# B&R Automation Studio project BaseProject (part 3)

#### AdvIecChk.st - Implementation file
```iecst
(*****************************************************************************************************************************************
- This library is not officially supported by
- Just like IECCheck library, this library only works IF a programming error was caused in a
program written in IEC languages.
This library will NOT help TO troubleshoot pagefaults caused in C, C++ etc.
- Automation Runtime Simulation (ArSim) does NOT provide consistent backtrace with this
library.
- This library is capable OF catching many types OF IEC programming errors but NOT all.
[Example: IF a pointer is NOT a null pointer but it is just pointing TO an incorrect but
NOT invalid OR protected location in the memory. The memory copy operation using
such pointer might end up overwriting some part OF the memory.
When the processor tries TO ACCESS this corrupted memory location, it will cause a
pagefault. In such cases, the memory has already been corrupted, so there are no
ways TO tell what wrote into this memory.]
 *****************************************************************************************************************************************
 * Library: AdvIecCheck
 ****************************************************************************************************************************************
 ****************************************************************************************************************************************
 *																																		*
 * 							How	to	isolate	pagefaults	using	the	 AdvIecCheck	library?											*
 *							~~~~~~~~~~~~~~~~~~~~~~~~~~~~~~~~~~~~~~~~~~~~~~~~~~~~~~~~~~~~~~~~											*
 ****************************************************************************************************************************************
 ****************************************************************************************************************************************

			1 Overview

					1.1 What is a pagefault (Processor Exception Error)?
					 While a system is running, if the processor is commanded TO ACCESS an invalid OR protected
					memory location, it throws an exception TO the operating system. The B&R operating system logs
					these types OF serious memory violation errors as pagefaults.

					1.2 What can cause a pagefault?
					 Pagefaults can be caused BY programming errors AND sometimes it can be very difficult TO
					FIND the root cause OF it. The programming errors, such as incorrect reads OR writes can be caused BY
					following reasons:
					- Null OR incorrect pointer handle
					- Division BY zero
					- Invalid range OF enumeration
					- Invalid index ACCESS OF an array

					1.3 What is the difference between IECcheck & AdvIecCheck library?
					The IEC check library which is provided with Automation Studio checks division BY zero, null pointer,
					invalid array index, invalid enumeration range ACCESS AND invalid subrange.
					- IF IECcheck is NOT added TO a project, the checks FOR ‘null OR incorrect pointer handle, division
					BY zero, invalid range OF enumeration, and invalid index ACCESS OF an array’ are NOT
					performed, but when pagefault is encountered, you will get a backtrace.
					This backtrace may point you TO the line OF code that might have caused the pagefault.
					- IF IECcheck is added TO a project, the checks FOR ‘null OR incorrect pointer handle, division BY
					zero, invalid range OF enumeration, and invalid index ACCESS OF an array’ are performed.
					IF the processor finds any OF those checks TO be incorrect, a logbook error entry will inform
					you what type OF error were found AND which task class caused it, but you will get NOT get a
					backtrace.
					The Advance IEC Check library performs the same basic functions as IEC Check, but it also provides
					the following additional data about the location OF the pagefault.
					- Last executed task class cyclic
					- Last executed task’s name
					- Type OF programming error
					- Variable values from the last executed line OF code
					- Backtrace pointing TO the last executed line OF code

			2 Required Software
					- Automation Studio 4 (or higher)
					- Automation Runtime Embedded OR Automation Runtime Windows

			3 **************************************Warning****************************************************
			  **************************************Warning****************************************************
					- Just like IECCheck library, this library only works IF a programming error was caused in a
					program written in IEC languages.
					This library will NOT help TO troubleshoot pagefaults caused in C, C++ etc.
					- Automation Runtime Simulation (ArSim) does NOT provide consistent backtrace with this
					library.
					- This library is capable OF catching many types OF IEC programming errors but NOT all.
					[Example: IF a pointer is NOT a null pointer but it is just pointing TO an incorrect but
					NOT invalid OR protected location in the memory. The memory copy operation using
					such pointer might end up overwriting some part OF the memory.
					When the processor tries TO ACCESS this corrupted memory location, it will cause a
					pagefault. In such cases, the memory has already been corrupted, so there are no
					ways TO tell what wrote into this memory.]
			   **************************************Warning****************************************************
			   **************************************Warning****************************************************

			4 How TO use the AdvIecCheck Library?
			  How TO FIND the cause OF a pagefault?
					1. Unzip the attached AdvIecChk library.
					2. Add this library TO the Automation Studio project that is causing a pagefault.
					 Help on adding a user library can be found at:
					 Automation Studio Help > Programming > Libraries >
					 Example: Creating a user library> Exporting AND importing libraries
					3. Make sure the newly added AdvIecChk library is inside software configuration > library objects.
					4. Re-build the project AND transfer it TO the target OR create new compact flash card.
					5. Wait FOR the pagefaults.
					6. Try TO have multiple pagefaults & a repeatable way TO reproduce them before opening the logbook
					inside the project.
					7. Sort the logbook BY TIME.
					8. Warning entry will give you the following information about the pagefault trapped BY AdvIecChk.
					- Task class cyclic OF the task (E.g. task class 4)
					- Name OF the task (E.g. PageFault was the name OF my task)
					- Type OF programming error (E.g. Unsigned Subrange was outside valid range)
					- MAX, min valid value OF the variable that caused this fault
					(The valid range FOR that USINT was [3..20] AND the element the program was trying TO ACCESS
					was at location 0.)
					- Value OF the variable that ended up causing this fault
					9. Click on the Error entry AND go TO the backtrace, double click on the ‘FUNCTION start position’ OF the
					task name that you found inside the last warning message (It is ‘Pagefault’ in my example).
					Wherever the Automation Studio takes you, it is the line OF code where the pagefault was
					encountered.
					 10. After fixing the code, repeat the steps that you used TO cause the pagefault AND make sure the
					programing error is resolved.

			5 How TO disable IecCheck OR AdvIecCheck library in the project?
					IF the option -D _IGNORE_CHECKLIB is enabled in the additional build options, then the functions
					in this library are NOT used otherwise even IF you DELETE this library from software configuration,
					the compiler will use it.

			6 Best practices TO catch a pagefault
					Check FOR the following types OF operations:
					- Memory set, move, copy, and compare
					- String set, move, copy, and compare
					- Loop, enumeration AND array ranges
					- Use OF ADR(), ACCESS, and pointer handles TO FUNCTION blocks

			7 Additional note
					- You can customize AdvIecChk library TO get even more customized information out OF it
					- IF a non IEC language is causing pagefault, declare a remanent variable AND increase value OF
					that variable in your program. After a pagefault, you can connect TO the target AND read the
					value OF that remanent variable. Find out, at which point you set that value in your code.
					The programming error should be after that line OF code.

 ***************************************************************************************************************************************
 ******************************************************Release Notes********************************************************************
Revision 1.00.0    - Matt Buck & Matt Adams
- Started distributing from 2013
- Better logger entries
 ******************************************************************************************************************************************
Revision 2.00.0    - Varad Darji
- Started distributing from Automation Conf. 2015
- Improvement for logger entries
- Provides backtrace
- gIecChkSec entries does NOT need TO be part OF this code there anymore because we are getting an actual backtrace now.
  They are there for legacy reasons.
- Created new documentation & added it to the library as well.
 ******************************************************************************************************************************************
 ******************************************************************************************************************************************)

(* Check divisor for DINT and UDINT division *)
FUNCTION CheckDivDWord
	IF divisor=0 THEN
		CheckDivDWord:=1;
		MakeEntry(55555,divisor,'Divide by Zero - Double Word');

		//Note: DarjiV, creating a pagefault on purpose to get the backtrace data
		//				This function does not provide consistant back
		memcpy(1,1,1);

	ELSE
		CheckDivDWord:=divisor;
	END_IF
END_FUNCTION

(* Check divisor for INT and UINT division *)
FUNCTION CheckDivWord
	IF divisor=0 THEN
		CheckDivWord:=1;
		MakeEntry(55555,divisor,'Divide by Zero - Word');

		//creating a pagefault on purpose to get the backtrace data
		memcpy(1,1,1);
	ELSE
		CheckDivWord:=divisor;
	END_IF
END_FUNCTION

(* Check divisor for SINT and USINT division *)
FUNCTION CheckDivByte
	IF divisor=0 THEN
		CheckDivByte:=1;
		MakeEntry(55555,divisor,'Divide by Zero - Byte');

		//creating a pagefault on purpose to get the backtrace data
		memcpy(1,1,1);
	ELSE
		CheckDivByte:=divisor;
	END_IF
END_FUNCTION

(* Check divisor for REAL division *)
FUNCTION CheckDivReal
	IF divisor=0 THEN
		CheckDivReal:=1;
		MakeEntry(55555,0,'Divide by Zero - Real');

		//creating a pagefault on purpose to get the backtrace data
		memcpy(1,1,1);
	ELSE
		CheckDivReal:=divisor;
	END_IF
END_FUNCTION

(* Check divisor for LREAL division *)
FUNCTION CheckDivLReal
	IF divisor=0 THEN
		CheckDivLReal:=1;
		MakeEntry(55555,0,'Divide by Zero - Long Real');

		//creating a pagefault on purpose to get the backtrace data
		memcpy(1,1,1);
	ELSE
		CheckDivLReal:=divisor;
	END_IF
END_FUNCTION

(* Check range for enumeration *)
FUNCTION CheckRange
	IF value < lower THEN
		CheckRange := lower;

		itoa(lower, ADR(LowString));
		itoa(upper, ADR(UpString));
		itoa(value, ADR(IndexString));
		strcpy(ADR(text),ADR('ENUM-Check Low. Value '));
		strcat(ADR(text),ADR(IndexString));
		strcat(ADR(text),ADR(' is outside ['));
		strcat(ADR(text),ADR(LowString));
		strcat(ADR(text),ADR('..'));
		strcat(ADR(text),ADR(UpString));
		strcat(ADR(text),ADR(']'));
		MakeEntry(55555,value,text);
		//creating a pagefault on purpose to get the backtrace data
		memcpy(1,1,1);

	ELSIF value > upper THEN
		CheckRange := upper;

		itoa(lower, ADR(LowString));
		itoa(upper, ADR(UpString));
		itoa(value, ADR(IndexString));
		strcpy(ADR(text),ADR('ENUM-Check High. Value '));
		strcat(ADR(text),ADR(IndexString));
		strcat(ADR(text),ADR(' is outside ['));
		strcat(ADR(text),ADR(LowString));
		strcat(ADR(text),ADR('..'));
		strcat(ADR(text),ADR(UpString));
		strcat(ADR(text),ADR(']'));
		MakeEntry(55555,value,text);
		//creating a pagefault on purpose to get the backtrace data
		memcpy(1,1,1);
	ELSE
		CheckRange := value;
	END_IF
END_FUNCTION

(* Check range for subrange of signed data types *)
FUNCTION CheckSignedSubrange
	IF value < lower THEN
		CheckSignedSubrange := lower;

		itoa(lower, ADR(LowString));
		itoa(upper, ADR(UpString));
		itoa(value, ADR(IndexString));
		strcpy(ADR(text),ADR('Signed Subrange Index '));
		strcat(ADR(text),ADR(IndexString));
		strcat(ADR(text),ADR(' is outside ['));
		strcat(ADR(text),ADR(LowString));
		strcat(ADR(text),ADR('..'));
		strcat(ADR(text),ADR(UpString));
		strcat(ADR(text),ADR(']'));
		MakeEntry(55555,value,text);
		//creating a pagefault on purpose to get the backtrace data
		memcpy(1,1,1);

	ELSIF value > upper THEN
		CheckSignedSubrange := upper;

		itoa(lower, ADR(LowString));
		itoa(upper, ADR(UpString));
		itoa(value, ADR(IndexString));
		strcpy(ADR(text),ADR('Signed Subrange Index '));
		strcat(ADR(text),ADR(IndexString));
		strcat(ADR(text),ADR(' is outside ['));
		strcat(ADR(text),ADR(LowString));
		strcat(ADR(text),ADR('..'));
		strcat(ADR(text),ADR(UpString));
		strcat(ADR(text),ADR(']'));
		MakeEntry(55555,value,text);
		//creating a pagefault on purpose to get the backtrace data
		memcpy(1,1,1);
	ELSE
		CheckSignedSubrange := value;
	END_IF
END_FUNCTION

(* Check range for subrange of unsigned data types *)
FUNCTION CheckUnsignedSubrange
	IF value < lower THEN
		CheckUnsignedSubrange := lower;

		itoa(lower, ADR(LowString));
		itoa(upper, ADR(UpString));
		itoa(value, ADR(IndexString));
		strcpy(ADR(text),ADR('Unsigned Subrange Index '));
		strcat(ADR(text),ADR(IndexString));
		strcat(ADR(text),ADR(' is outside ['));
		strcat(ADR(text),ADR(LowString));
		strcat(ADR(text),ADR('..'));
		strcat(ADR(text),ADR(UpString));
		strcat(ADR(text),ADR(']'));
		MakeEntry(55555,value,text);
		//creating a pagefault on purpose to get the backtrace data
		memcpy(1,1,1);

	ELSIF value > upper THEN
		CheckUnsignedSubrange := upper;

		itoa(lower, ADR(LowString));
		itoa(upper, ADR(UpString));
		itoa(value, ADR(IndexString));
		strcpy(ADR(text),ADR('Unsigned Subrange Index '));
		strcat(ADR(text),ADR(IndexString));
		strcat(ADR(text),ADR(' is outside ['));
		strcat(ADR(text),ADR(LowString));
		strcat(ADR(text),ADR('..'));
		strcat(ADR(text),ADR(UpString));
		strcat(ADR(text),ADR(']'));
		MakeEntry(55555,value,text);
		//creating a pagefault on purpose to get the backtrace data
		memcpy(1,1,1);
	ELSE
		CheckUnsignedSubrange := value;
	END_IF
END_FUNCTION

(* Check address when reading dynamic variables *)
FUNCTION CheckReadAccess
	IF address=0 THEN
		(* TODO: Insert an appropriate code, see AutomationStudio help for further information *)
		MakeEntry(55555,address,'Attempt to read from address of zero / NULL');
		//creating a pagefault on purpose to get the backtrace data
		memcpy(1,1,1);

	END_IF

	CheckReadAccess:=0;
END_FUNCTION

(* Check address when writing dynamic variables *)
FUNCTION CheckWriteAccess
	IF address=0 THEN
		(* TODO: Insert an appropriate code, see AutomationStudio help for further information *)
		MakeEntry(55555,address,'Attempt to write to address of zero / NULL');
		//creating a pagefault on purpose to get the backtrace data
		memcpy(1,1,1);
	END_IF

	CheckWriteAccess:=0;
END_FUNCTION

FUNCTION CheckBounds (* Check range for array access *)
	IF index < lower OR index > upper THEN
		itoa(lower, ADR(LowString));
		itoa(upper, ADR(UpString));
		itoa(index, ADR(IndexString));
		CheckBounds := upper;
		strcpy(ADR(text),ADR('Array Index '));
		strcat(ADR(text),ADR(IndexString));
		strcat(ADR(text),ADR(' is outside ['));
		strcat(ADR(text),ADR(LowString));
		strcat(ADR(text),ADR('..'));
		strcat(ADR(text),ADR(UpString));
		strcat(ADR(text),ADR(']'));
		MakeEntry(55555,index,text);
		//creating a pagefault on purpose to get the backtrace data
		memcpy(1,1,1);
	ELSE
		CheckBounds := index;
	END_IF
END_FUNCTION

FUNCTION MakeEntry (* Makes a log book entry. Note that gIecChkSec must be a global DINT! *)
	status_name := ST_name(0,ADR(taskname),ADR(group));
	PV_xgetadr(ADR('gIecChkSec'), ADR(pv_adr), ADR(data_len));
	IF pv_adr > 0 AND data_len > 0 THEN
		memcpy(ADR(SectionData),pv_adr,data_len);
		itoa(SectionData,ADR(SectionString));
	END_IF

	strcpy(ADR(out_text),ADR(text));
	strcat(ADR(out_text),ADR(' in task "'));
	strcat(ADR(out_text),ADR(taskname));
	strcat(ADR(out_text),ADR('" Section:'));
	strcat(ADR(out_text),ADR(SectionString));
	MakeEntry := ADR(out_text);

	// Making Logger entry & restarting
	ERRxwarning(number,index,ADR(out_text));
	// Change Note DarjiV: Change ERRxfatel_FB to ERRxwarning_FB because to get additional data.
	// 						Because I want TO finish this function and go back TO whichever function started this function and cause a pagefault there to get backtrace to the CODE.
	//						Now the AdvanceIEC Check library will give a pagefault location in CODE & the values of those variable when the pagefault happened.

END_FUNCTION
```

### Program Logical/Source/GlobalSetup (IEC)

#### Main.st
```iecst
PROGRAM _INIT
	(* Call global variables until they are use somewhere else *)
	gSampleTrak;
	gSampleTrak_SectorTrakA;
	gSampleTrak_SectorTrakB;
	gSampleTrak_SectorTrakAll;
	gSampleTrakMon;

	#ifdef ASSEMBLY_STANDARD
	(*All segment references must be included in the following segment array*)
	gTrakData.Seg.SegList[0].Name  := 'gSeg_A_1'; 		gTrakData.Seg.SegList[0].McType := gSeg_A_1 ;
	gTrakData.Seg.SegList[1].Name  := 'gSeg_A_2';		gTrakData.Seg.SegList[1].McType := gSeg_A_2 ;
	gTrakData.Seg.SegList[2].Name  := 'gSeg_A_3'; 		gTrakData.Seg.SegList[2].McType := gSeg_A_3 ;
	gTrakData.Seg.SegList[3].Name  := 'gSeg_A_4';		gTrakData.Seg.SegList[3].McType := gSeg_A_4 ;
	gTrakData.Seg.SegList[4].Name  := 'gSeg_A_5';		gTrakData.Seg.SegList[4].McType := gSeg_A_5 ;
	gTrakData.Seg.SegList[5].Name  := 'gSeg_A_6';		gTrakData.Seg.SegList[5].McType := gSeg_A_6 ;
	gTrakData.Seg.SegList[6].Name  := 'gSeg_A_7';		gTrakData.Seg.SegList[6].McType := gSeg_A_7 ;
	gTrakData.Seg.SegList[7].Name  := 'gSeg_A_8';		gTrakData.Seg.SegList[7].McType := gSeg_A_8 ;
	gTrakData.Seg.SegList[8].Name  := 'gSeg_A_9';		gTrakData.Seg.SegList[8].McType := gSeg_A_9 ;
	gTrakData.Seg.SegList[9].Name  := 'gSeg_A_10';		gTrakData.Seg.SegList[9].McType := gSeg_A_10;
	gTrakData.Seg.SegList[10].Name := 'gSeg_A_11';		gTrakData.Seg.SegList[10].McType := gSeg_A_11;
	gTrakData.Seg.SegList[11].Name := 'gSeg_A_12';		gTrakData.Seg.SegList[11].McType := gSeg_A_12;

	gTrakData.Seg.SegList[12].Name  := 'gSeg_B_1';		gTrakData.Seg.SegList[12].McType := gSeg_B_1;
	gTrakData.Seg.SegList[13].Name  := 'gSeg_B_2';		gTrakData.Seg.SegList[13].McType := gSeg_B_2;
	gTrakData.Seg.SegList[14].Name  := 'gSeg_B_3';		gTrakData.Seg.SegList[14].McType := gSeg_B_3;
	gTrakData.Seg.SegList[15].Name  := 'gSeg_B_4';		gTrakData.Seg.SegList[15].McType := gSeg_B_4;
	gTrakData.Seg.SegList[16].Name  := 'gSeg_B_5';		gTrakData.Seg.SegList[16].McType := gSeg_B_5;
	gTrakData.Seg.SegList[17].Name  := 'gSeg_B_6';		gTrakData.Seg.SegList[17].McType := gSeg_B_6;
	gTrakData.Seg.SegList[18].Name  := 'gSeg_B_7';		gTrakData.Seg.SegList[18].McType := gSeg_B_7;
	gTrakData.Seg.SegList[19].Name  := 'gSeg_B_8';		gTrakData.Seg.SegList[19].McType := gSeg_B_8;
	gTrakData.Seg.SegList[20].Name  := 'gSeg_B_9';		gTrakData.Seg.SegList[20].McType := gSeg_B_9;
	gTrakData.Seg.SegList[21].Name  := 'gSeg_B_10';		gTrakData.Seg.SegList[21].McType := gSeg_B_10;
	gTrakData.Seg.SegList[22].Name  := 'gSeg_B_11';		gTrakData.Seg.SegList[22].McType := gSeg_B_11;

	gTrakData.Seg.SegCount := 23;

	gTrakData.Seg.SegListAdr := ADR(gTrakData.Seg.SegList);

	#endif

END_PROGRAM

PROGRAM _CYCLIC
	(* Insert code here *)

END_PROGRAM

PROGRAM _EXIT
	(* Insert code here *)

END_PROGRAM
```

### Global.var
```iecst
VAR
	gTrakSystem : TrakType;
	gSampleTrakMon : McAcpTrakAssemblyMonData;
END_VAR
```

### Global.typ
```iecst
(*==================================================
ACOPOStrak Global Structure Hierarchy
==================================================*)

TYPE
	TrakType : 	STRUCT  (*Global structure definition*)
		Asm : TrBaseAsmType; (*Assembly substructure*)
		Par : TrakParametersType; (*ACOPOStrak application parameters*)
		Buffer : ARRAY[0..149]OF BOOL;
		Tracking : TrBaseTrackingType;
	END_STRUCT;
END_TYPE

(*Application parameters*)

TYPE
	TrakParametersType : 	STRUCT
		Velocity : REAL;
		Acceleration : REAL;
		CriticalVelocity : REAL;
		RecoveryVelocity : REAL;
	END_STRUCT;
END_TYPE

(*Interface for variable mapping*)

TYPE
	ModuleInterfaceType : 	STRUCT
		ShuttleMon : McAcpTrakAssemblyMonData;
		SampleTrak : McAssemblyType;
		MainPml : MpComIdentType;
		ModulePml : MpComIdentType;
		AlarmCore : MpComIdentType;
		AuditCore : MpComIdentType;
		RecipeCore : MpComIdentType;
		TrakInterface : TrakType;
		SectorTrakAll : McSectorType;
		SectorTrakB : McSectorType;
		SectorTrakA : McSectorType;
	END_STRUCT;
END_TYPE
```

### Program Logical/Source/TSM (IEC)

#### Main.st
```iecst
PROGRAM _INIT

END_PROGRAM

PROGRAM _CYCLIC
	(* Insert code here *)

	fbMainTsm(MpLink := ADR(gMainModule),
						Enable := TRUE,
						Parameters := ADR(parMainTsm));

	MpPackMLStateIsActive(gMainModule,mpPACKML_STATE_EXECUTE,1);
	gTrakSystem;
END_PROGRAM

PROGRAM _EXIT
	(* Insert code here *)

END_PROGRAM
```

### Program Logical/Source/TSMMain (IEC)

#### Main.st
```iecst
PROGRAM _INIT
	(* Insert code here *)

END_PROGRAM

PROGRAM _CYCLIC
	(* Call version control variables so they can be updated during every project build *)
	 MachineLastRevisionDate;
	 MachineSoftwareVersion;

END_PROGRAM

PROGRAM _EXIT
	(* Insert code here *)

END_PROGRAM
```

### Program Logical/Source/TSMAlarm (IEC)

#### Variables.var
```iecst
VAR
	fbAlarmMainTSM : MpAlarmXCore;
	FilterConfiguration : STRING[1000] := '';
	SortConfiguration : STRING[1000] := '';
	HistoryFilter : STRING[2000] := '';
	HistorySort : STRING[2000] := '';
	fbAlarmHistMainTSM : MpAlarmXHistory;
	TriggerTestAlarm : BOOL;
END_VAR
```

#### Main.st
```iecst
PROGRAM _INIT
	(* Insert code here *)
	FilterConfiguration;
	SortConfiguration;
	HistoryFilter;
	HistorySort;
END_PROGRAM

PROGRAM _CYCLIC
	(* Insert code here *)
	fbAlarmMainTSM(MpLink := ADR(gAlarmXCore), Enable := TRUE);
	fbAlarmHistMainTSM(MpLink := ADR(gAlarmXHistory), Enable := TRUE, DeviceName := ADR('User'));

	// Reset the Export cmd from mappView when export is done
	IF fbAlarmHistMainTSM.Export AND fbAlarmHistMainTSM.CommandDone THEN
		fbAlarmHistMainTSM.Export := FALSE;
	END_IF

	TriggerTestAlarm;

END_PROGRAM

PROGRAM _EXIT
	(* Insert code here *)

END_PROGRAM
```

### TrakDiagGlobal.var
```iecst
(*LogBook variables*)
VAR
	LogbookInterface : LogBookCtrlType; (*Logbook main structure*)
END_VAR
VAR CONSTANT
	LOGBOOK_EXECUTIONS : USINT := 10; (*Executions per cycle*)
	LOGBOOK_ENTRIES_MAX : UINT := 100; (*Total number of entries*)
	LOGBOOK_BOOKS_MAX : USINT := 13; (*Total number of facilities*)
	LOGBOOK_TEXT_LEN : UINT := 200; (*Error text length*)
END_VAR
(*Module definitions*)
VAR
	DiagInterface : ModuleInterfaceType;
	ModuleName : STRING[40];
END_VAR
```

### Program Logical/Source/Diagnostic/DiagConfig (IEC)

#### Init.st - Init code
```iecst
PROGRAM _INIT
	(* Insert code here *)

		(* Insert code here *)
	ModuleName := 'DiagModule';

	gRecipeXml_DiagModule;

END_PROGRAM
```

### Program Logical/Source/Diagnostic/DiagAlarm (IEC)

#### Main.st
```iecst
PROGRAM _INIT
	(* Insert code here *)
	FilterConfiguration;
	SortConfiguration;
	HistoryFilter;
	HistorySort;
	gAlarmXCore_DiagModule;

END_PROGRAM

PROGRAM _CYCLIC
	(* Insert code here *)

	fbAlarmDiagModule(MpLink := ADR(DiagInterface.AlarmCore), Enable := TRUE);

	TriggerTestAlarm;
	TriggerTestInformation;
	TriggerTestWarning;

END_PROGRAM

PROGRAM _EXIT
	(* Insert code here *)

END_PROGRAM
```

### Program Logical/Source/Diagnostic/TrakDiag (IEC)

#### Types.typ
```iecst
TYPE
	VisType : 	STRUCT
		OpenSegDialog : BOOL;
		OpenShuttleDialog : BOOL;
	END_STRUCT;
	CheckStateEnum :
		(
		WAIT_FOR_CHECK,
		READ_DATA,
		READ_DATA_SEG_STATE,
		CHECK_SEG_STATE,
		READ_DATA_SEG_ERROR_STAT,
		CHECK_ERROR_STAT,
		READ_DATA_SEG_ERROR,
		CHECK_ERROR_CODE,
		WRITE_WARNING_CODE,
		READ_DATA_SEG_LAG,
		CHECK_SEG_LAG,
		READ_DATA_SEG_VEL,
		CHECK_SEG_VEL,
		READ_DATA_SEG_TEMP,
		CHECK_DATA_SEG_TEMP,
		WRITE_SPEED_FILTER,
		WRITE_SPEED_FILTER_WAIT,
		WRITE_ZERO_PITCH,
		READ_EXEC_ERROR,
		READ_SEG_STATUS,
		WRITE_SEG_RESET,
		WAIT_FOR_DONE
		);
	SegErrorCheckType : 	STRUCT
		CheckState : CheckStateEnum;
		CmdCheckErrorCode : BOOL;
		DataReadExecutionError : BOOL;
		ErrorNumber : UINT;
		SegStatusBits : UDINT;
		ErrorStatusBit : BOOL;
		ErrorStatus : UDINT;
	END_STRUCT;
	DiagFbsType : 	STRUCT
		Asm : DiagAsmFbsTyp;
		Seg : DiagSegFbsTyp;
	END_STRUCT;
	DiagAsmFbsTyp : 	STRUCT
		ReadInfo : MC_BR_AsmReadInfo_AcpTrak;
		ReadStatus : MC_BR_AsmReadStatus_AcpTrak;
	END_STRUCT;
	DiagSegFbsTyp : 	STRUCT
		ReadInfo : ARRAY[0..NUM_SEG]OF MC_BR_SegReadInfo_AcpTrak;
		ReadStatus : ARRAY[0..NUM_SEG]OF MC_BR_SegReadStatus_AcpTrak;
		ProcessParID : ARRAY[0..NUM_SEG]OF MC_BR_SegProcessParID_AcpTrak;
	END_STRUCT;
END_TYPE
```

#### Variables.var
```iecst
VAR
	MC_BR_ShCopyUserData_AcpTrak_0 : MC_BR_ShCopyUserData_AcpTrak;
	ErrorCodeIDInfo : ARRAY[0..NUM_SEG] OF McAcpTrakSegProcessParIDType;
	SegWarningCmdIDInfo : McAcpTrakSegProcessParIDType;
	SegErrorCheck : ARRAY[0..NUM_SEG] OF SegErrorCheckType;
	CpuSim : BOOL;
END_VAR
(*For testing only*)
VAR
	MC_BR_SegCommandError_AcpTrak_0 : MC_BR_SegCommandError_AcpTrak;
END_VAR
(*Declarations for TrakMap*)
VAR
	paperCore : TrkPaperCore;
	paperOptions : TrkPaperCoreOptionsType;
	TrakDiag : TrkDiagStatusType;
	DiagFbs : DiagFbsType;
	SegIndex : USINT;
END_VAR
(******************* BE SURE TO CHANGE THIS TO MATCH YOUR OWN USER DATA TYPE!!! This is just set for the moment as an example user data type that likely won't exist in your project!*)
VAR
	ShuttleUserData : ShuttleUserDataType;
END_VAR
```

#### Cyclic.st
```iecst
PROGRAM _CYCLIC

	MC_BR_SegCommandError_AcpTrak_0(Segment := ADR(TrakDiag.Seg.SegList[0].McType));

	IF MC_BR_SegCommandError_AcpTrak_0.Done THEN
		MC_BR_SegCommandError_AcpTrak_0.Execute := FALSE;
	END_IF

	(***********************************ASSEMBLY INFORMATION******************************	)
	(*Read Assebly Status*)

	DiagFbs.Asm.ReadStatus.Enable	:= TRUE;
	DiagFbs.Asm.ReadStatus();

	IF DiagFbs.Asm.ReadStatus.Valid THEN
		TrakDiag.Asm.AssemblyDisabled 	:= DiagFbs.Asm.ReadStatus.AssemblyDisabled;
		TrakDiag.Asm.AssemblyErrorStop := DiagFbs.Asm.ReadStatus.AssemblyErrorStop;
		TrakDiag.Asm.AssemblyReady		:= DiagFbs.Asm.ReadStatus.AssemblyReady;
		TrakDiag.Asm.AssemblyHoming	:= DiagFbs.Asm.ReadStatus.AssemblyHoming;
		TrakDiag.Asm.AssemblyStopping	:= DiagFbs.Asm.ReadStatus.AssemblyStopping;
	END_IF

	(*Read Assembly Info *)

	DiagFbs.Asm.ReadInfo.Enable		:= TRUE;
	DiagFbs.Asm.ReadInfo();

	IF DiagFbs.Asm.ReadInfo.Valid THEN
		TrakDiag.Asm.CommunicationReady 	:= DiagFbs.Asm.ReadInfo.AssemblyInfo.CommunicationReady;
		TrakDiag.Asm.PowerOn				:= DiagFbs.Asm.ReadInfo.AssemblyInfo.PowerOn;
		TrakDiag.Asm.ReadyForPowerOn		:= DiagFbs.Asm.ReadInfo.AssemblyInfo.ReadyForPowerOn;
		TrakDiag.Asm.ShuttlesCount 			:= DiagFbs.Asm.ReadInfo.AssemblyInfo.ShuttlesCount;
		TrakDiag.Asm.ShuttleInErrorStopCount := DiagFbs.Asm.ReadInfo.AssemblyInfo.ShuttlesInErrorStopCount;
		TrakDiag.Asm.StartupCount			:= DiagFbs.Asm.ReadInfo.AssemblyInfo.StartupCount;
	END_IF

	(****************************** SEGMENT ERROR INFORMATION *****************************************)

	FOR SegIndex := 0 TO NUM_SEG DO

		IF TrakDiag.Seg.SegList[SegIndex].McType.controlif <> 0 THEN //If the array contains a segment reference

			DiagFbs.Seg.ReadInfo[SegIndex].Segment 	:= ADR(TrakDiag.Seg.SegList[SegIndex].McType);
			DiagFbs.Seg.ReadInfo[SegIndex].Enable	:= TRUE;
			DiagFbs.Seg.ReadInfo[SegIndex]();

			IF DiagFbs.Seg.ReadInfo[SegIndex].Valid THEN
				//Capture Segment Info
				TrakDiag.Seg.SegList[SegIndex].Status.CommunicationReady 	:= DiagFbs.Seg.ReadInfo[SegIndex].SegmentInfo.CommunicationReady;
				TrakDiag.Seg.SegList[SegIndex].Status.ReadyForPowerOn		:= DiagFbs.Seg.ReadInfo[SegIndex].SegmentInfo.ReadyForPowerOn;
				TrakDiag.Seg.SegList[SegIndex].Status.PowerOn				:= DiagFbs.Seg.ReadInfo[SegIndex].SegmentInfo.PowerOn;
				TrakDiag.Seg.SegList[SegIndex].Status.StartupCount			:= DiagFbs.Seg.ReadInfo[SegIndex].SegmentInfo.StartupCount;
				TrakDiag.Seg.SegList[SegIndex].Status.CommunicationState	:= DiagFbs.Seg.ReadInfo[SegIndex].SegmentInfo.CommunicationState;

			END_IF

			DiagFbs.Seg.ReadStatus[SegIndex].Segment := ADR(TrakDiag.Seg.SegList[SegIndex].McType);
			DiagFbs.Seg.ReadStatus[SegIndex].Enable	:= TRUE;
			DiagFbs.Seg.ReadStatus[SegIndex]();

			IF DiagFbs.Seg.ReadStatus[SegIndex].Valid THEN

				//Check for change of state to ErrorStop to command reading error data, IF communication is ready
				IF ((TrakDiag.Seg.SegList[SegIndex].Status.SegmentErrorStop = FALSE AND DiagFbs.Seg.ReadStatus[SegIndex].SegmentErrorStop = TRUE))
					AND (TrakDiag.Seg.SegList[SegIndex].Status.CommunicationReady = TRUE) THEN

					SegErrorCheck[SegIndex].CmdCheckErrorCode := TRUE;

					//Check for change of state from ErrorStop to reset error number in diag structure
				ELSIF ((TrakDiag.Seg.SegList[SegIndex].Status.SegmentErrorStop = TRUE) AND (DiagFbs.Seg.ReadStatus[SegIndex].SegmentErrorStop = FALSE))
					AND (TrakDiag.Seg.SegList[SegIndex].Status.CommunicationReady = TRUE) THEN

					TrakDiag.Seg.SegList[SegIndex].Status.ErrorCode := 0;

				END_IF
				//Capture Segment Status

				TrakDiag.Seg.SegList[SegIndex].Status.SegmentDisabled	:= DiagFbs.Seg.ReadStatus[SegIndex].SegmentDisabled;
				TrakDiag.Seg.SegList[SegIndex].Status.SegmentErrorStop	:= DiagFbs.Seg.ReadStatus[SegIndex].SegmentErrorStop;
				TrakDiag.Seg.SegList[SegIndex].Status.SegmentReady		:= DiagFbs.Seg.ReadStatus[SegIndex].SegmentReady;
				TrakDiag.Seg.SegList[SegIndex].Status.SegmentStopping	:= DiagFbs.Seg.ReadStatus[SegIndex].SegmentStopping;
			END_IF
		END_IF
	END_FOR

	CpuSim := DiagCpuIsSimulated() OR DiagCpuIsARsim();

	IF CpuSim = FALSE THEN
		actCheckErrorCode;
	END_IF

	(***********************************TRAKMAP******************************)

	//Fetch ShuttleUserData Example

	(* This will likely change to match your project! This is just an example of how to use the
		the click to get a shuttle's user data. The inputs to the ShCopyUserData will reflect your own project
	*)
//	IF EDGEPOS(paperCore.ClickData.Shuttle.Valid) THEN
//		MC_BR_ShCopyUserData_AcpTrak_0.Axis         := ADR(paperCore.ClickData.Shuttle.Data.Axis);
//		MC_BR_ShCopyUserData_AcpTrak_0.Execute      := TRUE;
//		MC_BR_ShCopyUserData_AcpTrak_0.DataAddress  := ADR(ShuttleUserData);
//		MC_BR_ShCopyUserData_AcpTrak_0.DataSize     := SIZEOF(ShuttleUserData);
//		MC_BR_ShCopyUserData_AcpTrak_0.Mode         := mcACPTRAK_USERDATA_GET;
//	END_IF

	paperCore();

	MC_BR_ShCopyUserData_AcpTrak_0();
	MC_BR_ShCopyUserData_AcpTrak_0.Execute := FALSE;

END_PROGRAM
```

#### Init.st
```iecst
PROGRAM _INIT

	SegDefinition;

	paperCore.SegmentCount := TrakDiag.Seg.SegCount;
	paperCore.Segments := ADR(TrakDiag.Seg.SegList);
	paperCore.Options := ADR(paperOptions);
	paperCore.Enable := TRUE;

END_PROGRAM
```

#### SegDefinition.st
```iecst
//This file was automatically generated using the TrakMapImporter program. Verify that the segment names and assembly name match your project values correctly
ACTION SegDefinition:
//	TrakDiag.Seg.SegList[0].Name  := 'gSeg_A_1';		TrakDiag.Seg.SegList[0].McType := gSeg_A_1;
//	TrakDiag.Seg.SegList[1].Name  := 'gSeg_A_2';		TrakDiag.Seg.SegList[1].McType := gSeg_A_2;
//	TrakDiag.Seg.SegList[2].Name  := 'gSeg_A_3';		TrakDiag.Seg.SegList[2].McType := gSeg_A_3;
//	TrakDiag.Seg.SegList[3].Name  := 'gSeg_A_4';		TrakDiag.Seg.SegList[3].McType := gSeg_A_4;
//	TrakDiag.Seg.SegList[4].Name  := 'gSeg_A_5';		TrakDiag.Seg.SegList[4].McType := gSeg_A_5;
//	TrakDiag.Seg.SegList[5].Name  := 'gSeg_A_6';		TrakDiag.Seg.SegList[5].McType := gSeg_A_6;
//	TrakDiag.Seg.SegList[6].Name  := 'gSeg_A_7';		TrakDiag.Seg.SegList[6].McType := gSeg_A_7;
//	TrakDiag.Seg.SegList[7].Name  := 'gSeg_A_8';		TrakDiag.Seg.SegList[7].McType := gSeg_A_8;
//	TrakDiag.Seg.SegList[8].Name  := 'gSeg_A_9';		TrakDiag.Seg.SegList[8].McType := gSeg_A_9;
//	TrakDiag.Seg.SegList[9].Name  := 'gSeg_A_10';		TrakDiag.Seg.SegList[9].McType := gSeg_A_10;
//	TrakDiag.Seg.SegList[10].Name  := 'gSeg_A_11';		TrakDiag.Seg.SegList[10].McType := gSeg_A_11;
//	TrakDiag.Seg.SegList[11].Name  := 'gSeg_A_12';		TrakDiag.Seg.SegList[11].McType := gSeg_A_12;
//	TrakDiag.Seg.SegList[12].Name  := 'gSeg_B_1';		TrakDiag.Seg.SegList[12].McType := gSeg_B_1;
//	TrakDiag.Seg.SegList[13].Name  := 'gSeg_B_2';		TrakDiag.Seg.SegList[13].McType := gSeg_B_2;
//	TrakDiag.Seg.SegList[14].Name  := 'gSeg_B_3';		TrakDiag.Seg.SegList[14].McType := gSeg_B_3;
//	TrakDiag.Seg.SegList[15].Name  := 'gSeg_B_4';		TrakDiag.Seg.SegList[15].McType := gSeg_B_4;
//	TrakDiag.Seg.SegList[16].Name  := 'gSeg_B_5';		TrakDiag.Seg.SegList[16].McType := gSeg_B_5;
//	TrakDiag.Seg.SegList[17].Name  := 'gSeg_B_6';		TrakDiag.Seg.SegList[17].McType := gSeg_B_6;
//	TrakDiag.Seg.SegList[18].Name  := 'gSeg_B_7';		TrakDiag.Seg.SegList[18].McType := gSeg_B_7;
//	TrakDiag.Seg.SegList[19].Name  := 'gSeg_B_8';		TrakDiag.Seg.SegList[19].McType := gSeg_B_8;
//	TrakDiag.Seg.SegList[20].Name  := 'gSeg_B_9';		TrakDiag.Seg.SegList[20].McType := gSeg_B_9;
//	TrakDiag.Seg.SegList[21].Name  := 'gSeg_B_10';		TrakDiag.Seg.SegList[21].McType := gSeg_B_10;
//	TrakDiag.Seg.SegList[22].Name  := 'gSeg_B_11';		TrakDiag.Seg.SegList[22].McType := gSeg_B_11;

	TrakDiag.Seg.SegCount := 23;

	TrakDiag.Seg.SegListAdr := ADR(TrakDiag.Seg.SegList);

	DiagFbs.Asm.ReadInfo.Assembly := ADR(gSampleTrak);
	DiagFbs.Asm.ReadStatus.Assembly := ADR(gSampleTrak);

	paperCore.ViewBoxCfg.MinX := -0.735577;
	paperCore.ViewBoxCfg.MinY := -0.115;
	paperCore.ViewBoxCfg.Width := 2.13115;
	paperCore.ViewBoxCfg.Height := 1.52;
END_ACTION
```

### Program Logical/Source/Diagnostic/Logbook (IEC)

#### Types.typ
```iecst
TYPE
	LogBooksType : 	STRUCT
		Ident : ARRAY[0..LOGBOOK_BOOKS_MAX]OF UDINT;
		RecordIDLatest : ARRAY[0..LOGBOOK_BOOKS_MAX]OF UDINT;
		RecordIDOld : ARRAY[0..LOGBOOK_BOOKS_MAX]OF UDINT;
		RecordIDIsLast : ARRAY[0..LOGBOOK_BOOKS_MAX]OF BOOL;
		RecordID : ARRAY[0..LOGBOOK_BOOKS_MAX]OF UDINT;
		CntLogbook : USINT;
	END_STRUCT;
END_TYPE
```

#### Variables.var
```iecst
(*---------------------------------------------------------------------------------------------------------------------------------*)
VAR
	ErrorText : STRING[LOGBOOK_TEXT_LEN];
	cntFilterNo : UINT;
	cntFilterText : UINT;
	cntFilterLogbook : UINT;
	cntFilterSeverity : UINT;
	cntFilterDate : UINT;
	tmpSTR : STRING[100];
	tmpDT : DATE_AND_TIME;
	tmpDTstruct : DTStructure;
	TimeStart : DATE_AND_TIME;
	TimeEnd : DATE_AND_TIME;
	AddData : ARRAY[0..500] OF USINT;
	Logbook : LogBooksType;
	idx : UINT;
	eventID : DINT;
	animation : USINT;
END_VAR
(*---------------------------------------------------------------------------------------------------------------------------------*)
(*Local function*)
VAR
	ArEventLogGetPreviousRecordID_0 : ArEventLogGetPreviousRecordID;
	ArEventLogGetLatestRecordID_0 : ArEventLogGetLatestRecordID;
	ArEventLogRead_0 : ArEventLogRead;
	ArEventLogWrite_0 : ArEventLogWrite;
	ArEventLogReadErrorNumber_0 : ArEventLogReadErrorNumber;
	ArEventLogReadDescription_0 : ArEventLogReadDescription;
	ArEventLogReadAddData_0 : ArEventLogReadAddData;
	ArEventLogReadObjectID_0 : ArEventLogReadObjectID;
	DTGetTime_0 : DTGetTime;
	httpUtf8ToString_0 : httpUtf8ToString;
	AutoRefresh : TON_10ms;
END_VAR
(*Local variables*)
VAR
	LogbookState : LogBookStateEnum;
	ArEventLogGetIdent_0 : ArEventLogGetIdent;
	executions : USINT;
END_VAR
(*---------------------------------------------------------------------------------------------------------------------------------*)
(*Local constants*)
VAR CONSTANT
	LOGBOOK_NAMES : ARRAY[0..LOGBOOK_BOOKS_MAX] OF STRING[50] := ['$$accsec','$$diag','$$arlogconn','$$fieldbus','$$firewall','$$mapp','$$motion','$$safety','$$arlogsys','$$textsys','$$unitsys','$$arlogusr','$$vision','$$visu'];
	LOGBOOK_TEXT : ARRAY[0..LOGBOOK_BOOKS_MAX] OF STRING[50] := ['Access','Commissioning','Connectivity','Fieldbus','Firewall','Mapp','Motion','Safety','System','Text System','Unit System','User','Vision','Visualization'];
	NO_SPACE : UINT := 0;
END_VAR
(*read & filter motion logger*)
VAR
	EventID : DINT := 0;
	EventIDSeverity : USINT := 0;
	EventIDFacility : UINT := 0;
	EventIDCode : UINT := 0;
	EventTimeStamp : ArEventLogTimeStampType := (0);
	ObjectID : STRING[36] := '';
	Description : STRING[256] := '';
	TempString : STRING[32] := '';
	SegmentErrorFound : USINT := 0;
	AlarmCount : ARRAY[0..119] OF UDINT;
	TimeStruct : TIMEStructure;
	FirstEntryCheckSum : USINT;
END_VAR
```

#### LocalFunctions.st
```iecst
// --------------------------------------------------------------------------------------------------------------------
// Gets severity from EventId (bits 31-30)
FUNCTION GetSeverity
	IF ArEventLogIsError(EventID := EventID) THEN
		GetSeverity := arEVENTLOG_SEVERITY_ERROR;
	ELSIF ArEventLogIsWarning(EventID := EventID) THEN
		GetSeverity := arEVENTLOG_SEVERITY_WARNING;
	ELSIF ArEventLogIsInformation(EventID := EventID) THEN
		GetSeverity := arEVENTLOG_SEVERITY_INFO;
	ELSIF ArEventLogIsSuccess(EventID := EventID) THEN
		GetSeverity := arEVENTLOG_SEVERITY_SUCCESS;
	END_IF
END_FUNCTION

// --------------------------------------------------------------------------------------------------------------------
// Gets code from EventId (bits 15-0)
FUNCTION GetCode
	GetCode := DINT_TO_UINT(EventID);
END_FUNCTION

// --------------------------------------------------------------------------------------------------------------------
// Gets facility from EventId (bits 27-16)
FUNCTION GetFacility
	GetFacility := DINT_TO_UINT(SHR(EventID, 16) AND 16#0FFF);
END_FUNCTION

// --------------------------------------------------------------------------------------------------------------------
// --------------------------------------------------------------------------------------------------------------------
// Insert new entry
FUNCTION InsertEntry
	// Lets see where new entry fits
	FOR idx:=1 TO Data.EntriesTotal DO
		// Sorting is ascending
		IF Sorting = SORTING_ASC THEN
			// New entry is old than this entry
			IF DTsec < Data.Entries.DTsec[idx] THEN
				EXIT;
				// If entries are within the same second check milisecond data
			ELSIF DTsec = Data.Entries.DTsec[idx] THEN
				IF DTmsec < Data.Entries.DTmsec[idx] THEN
					EXIT;
				END_IF
			END_IF
			// Sorting is descending
		ELSE
			// New entry is newer than this entry
			IF DTsec > Data.Entries.DTsec[idx] THEN
				EXIT;
				// If entries are within the same second check milisecond data
			ELSIF DTsec = Data.Entries.DTsec[idx] THEN
				IF DTmsec > Data.Entries.DTmsec[idx] THEN
					EXIT;
				END_IF
			END_IF
		END_IF
	END_FOR;

	// Add data as long as buffer is not full
	IF Data.EntriesTotal < LOGBOOK_ENTRIES_MAX THEN
		IF Data.EntriesTotal = 1 AND idx = 1 THEN
			idy := 1;
		ELSIF Data.EntriesTotal >= idx THEN
			idy := Data.EntriesTotal - idx + 1;
		END_IF
		Data.EntriesTotal := Data.EntriesTotal + 1;
		// If buffer is full check where entry fits
	ELSE
		// Entry is beyond scope of buffer
		IF idx > LOGBOOK_ENTRIES_MAX THEN
			InsertEntry := NO_SPACE;
			RETURN;
		ELSE
			IF Data.EntriesTotal - idx > 0 THEN
				idy := Data.EntriesTotal - idx;
			END_IF
		END_IF
	END_IF

	// Dont move if there is nothing to move
	IF idy <> 0 THEN
		brsmemmove(ADR(Data.Entries.Code[idx+1]),ADR(Data.Entries.Code[idx]), idy * SIZEOF(Data.Entries.Code[1]));
		brsmemmove(ADR(Data.Entries.Timestamp[idx+1]),ADR(Data.Entries.Timestamp[idx]), idy * SIZEOF(Data.Entries.Timestamp[1]));
		brsmemmove(ADR(Data.Entries.DTsec[idx+1]),ADR(Data.Entries.DTsec[idx]), idy * SIZEOF(Data.Entries.DTsec[1]));
		brsmemmove(ADR(Data.Entries.DTmsec[idx+1]),ADR(Data.Entries.DTmsec[idx]), idy * SIZEOF(Data.Entries.DTmsec[1]));
		brsmemmove(ADR(Data.Entries.ErrorNo[idx+1]),ADR(Data.Entries.ErrorNo[idx]), idy * SIZEOF(Data.Entries.ErrorNo[1]));
		brsmemmove(ADR(Data.Entries.ErrorText[idx+1]),ADR(Data.Entries.ErrorText[idx]), idy * SIZEOF(Data.Entries.ErrorText[1]));
		brsmemmove(ADR(Data.Entries.EventID[idx+1]),ADR(Data.Entries.EventID[idx]), idy * SIZEOF(Data.Entries.EventID[1]));
		brsmemmove(ADR(Data.Entries.FacilityCode[idx+1]),ADR(Data.Entries.FacilityCode[idx]), idy * SIZEOF(Data.Entries.FacilityCode[1]));
		brsmemmove(ADR(Data.Entries.LogbookName[idx+1]),ADR(Data.Entries.LogbookName[idx]), idy * SIZEOF(Data.Entries.LogbookName[1]));
		brsmemmove(ADR(Data.Entries.Severity[idx+1]),ADR(Data.Entries.Severity[idx]), idy * SIZEOF(Data.Entries.Severity[1]));
	END_IF
	InsertEntry := idx;

END_FUNCTION

// --------------------------------------------------------------------------------------------------------------------
// Normalize 2 digit date and time values
FUNCTION NormalizeDateTime
	tmpSTR2 := AddSTR;
	IF(Value < 10) THEN
		brsstrcat(ADR(tmpSTR2), ADR('0'));
	END_IF
	brsitoa(Value, ADR(tmpSTR1));
	brsstrcat(ADR(tmpSTR2), ADR(tmpSTR1));
	brsstrcat(Target, ADR(tmpSTR2));
	NormalizeDateTime := TRUE;
END_FUNCTION

// --------------------------------------------------------------------------------------------------------------------
// Working status
FUNCTION WorkingStatus
	Animation := Animation+1;

	IF (Animation = 80) THEN
		Animation := 0;
	END_IF

	brsstrcpy(Target, Text);
	CASE(Animation) OF
		0..19	: brsstrcat(Target, ADR('/'));
		20..39	: brsstrcat(Target, ADR('-'));
		40..59	: brsstrcat(Target, ADR('\'));
		60..79	: brsstrcat(Target, ADR('|'));
	END_CASE;
	WorkingStatus := Animation;
END_FUNCTION

// --------------------------------------------------------------------------------------------------------------------
// Is second string in first string
FUNCTION IsInstr
	IF (brsstrlen(String1) > brsstrlen(String2)) THEN
		FOR idx:=0 TO brsstrlen(String1) - brsstrlen(String2) DO
			IF (brsmemcmp(String1 + idx, String2, brsstrlen(String2)) = 0) THEN
				IsInstr := TRUE;
				EXIT;
			END_IF
		END_FOR;
	END_IF
END_FUNCTION

(* Trigger proper alarms *)
FUNCTION SetTrakSegAlarm

		SetTrakSegAlarm := TRUE;
		// EventIDCode add new alarms triggers at the end otherwise
		// the AlarmCount has to be adjusted not just here but also for all the alarms in the MpAlarmX config

		CASE EventIDCode OF
		// every time the alarm is triggered it's counted so a total count can be displayed in the alarm message
		1	 :  AlarmCount[0  ] :=  AlarmCount[0]  + 1;   MpAlarmXSet(AlarmMpLink,'EventIDCode.1	');
		2	 :  AlarmCount[1  ] :=  AlarmCount[1]  + 1;   MpAlarmXSet(AlarmMpLink,'EventIDCode.2	');
		7	 :  AlarmCount[2  ] :=  AlarmCount[2]  + 1;   MpAlarmXSet(AlarmMpLink,'EventIDCode.7	');
		2048 :  AlarmCount[3  ] :=  AlarmCount[3]  + 1;   MpAlarmXSet(AlarmMpLink,'EventIDCode.2048');
		2049 :  AlarmCount[4  ] :=  AlarmCount[4]  + 1;   MpAlarmXSet(AlarmMpLink,'EventIDCode.2049');
		2050 :  AlarmCount[5  ] :=  AlarmCount[5]  + 1;   MpAlarmXSet(AlarmMpLink,'EventIDCode.2050');
		2051 :  AlarmCount[6  ] :=  AlarmCount[6]  + 1;   MpAlarmXSet(AlarmMpLink,'EventIDCode.2051');
		2052 :  AlarmCount[7  ] :=  AlarmCount[7]  + 1;   MpAlarmXSet(AlarmMpLink,'EventIDCode.2052');
		2053 :  AlarmCount[8  ] :=  AlarmCount[8]  + 1;   MpAlarmXSet(AlarmMpLink,'EventIDCode.2053');
		2054 :  AlarmCount[9  ] :=  AlarmCount[9]  + 1;   MpAlarmXSet(AlarmMpLink,'EventIDCode.2054');
		2055 :  AlarmCount[10 ] := AlarmCount[10]  + 1;   MpAlarmXSet(AlarmMpLink,'EventIDCode.2055');
		2056 :  AlarmCount[11 ] := AlarmCount[11]  + 1;   MpAlarmXSet(AlarmMpLink,'EventIDCode.2056');
		2057 :  AlarmCount[12 ] := AlarmCount[12]  + 1;   MpAlarmXSet(AlarmMpLink,'EventIDCode.2057');
		2058 :  AlarmCount[13 ] := AlarmCount[13]  + 1;   MpAlarmXSet(AlarmMpLink,'EventIDCode.2058');
		2060 :  AlarmCount[14 ] := AlarmCount[14]  + 1;   MpAlarmXSet(AlarmMpLink,'EventIDCode.2060');
		2061 :  AlarmCount[15 ] := AlarmCount[15]  + 1;   MpAlarmXSet(AlarmMpLink,'EventIDCode.2061');
		2063 :  AlarmCount[16 ] := AlarmCount[16]  + 1;   MpAlarmXSet(AlarmMpLink,'EventIDCode.2063');
		2064 :  AlarmCount[17 ] := AlarmCount[17]  + 1;   MpAlarmXSet(AlarmMpLink,'EventIDCode.2064');
		2066 :  AlarmCount[18 ] := AlarmCount[18]  + 1;   MpAlarmXSet(AlarmMpLink,'EventIDCode.2066');
		2067 :  AlarmCount[19 ] := AlarmCount[19]  + 1;   MpAlarmXSet(AlarmMpLink,'EventIDCode.2067');
		2068 :  AlarmCount[20 ] := AlarmCount[20]  + 1;   MpAlarmXSet(AlarmMpLink,'EventIDCode.2068');
		2069 :  AlarmCount[21 ] := AlarmCount[21]  + 1;   MpAlarmXSet(AlarmMpLink,'EventIDCode.2069');
		2070 :  AlarmCount[22 ] := AlarmCount[22]  + 1;   MpAlarmXSet(AlarmMpLink,'EventIDCode.2070');
		2071 :  AlarmCount[23 ] := AlarmCount[23]  + 1;   MpAlarmXSet(AlarmMpLink,'EventIDCode.2071');
		2074 :  AlarmCount[24 ] := AlarmCount[24]  + 1;   MpAlarmXSet(AlarmMpLink,'EventIDCode.2074');
		2077 :  AlarmCount[25 ] := AlarmCount[25]  + 1;   MpAlarmXSet(AlarmMpLink,'EventIDCode.2077');
		2080 :  AlarmCount[26 ] := AlarmCount[26]  + 1;   MpAlarmXSet(AlarmMpLink,'EventIDCode.7392');
		2082 :  AlarmCount[27 ] := AlarmCount[27]  + 1;   MpAlarmXSet(AlarmMpLink,'EventIDCode.2080');
		2083 :  AlarmCount[28 ] := AlarmCount[28]  + 1;   MpAlarmXSet(AlarmMpLink,'EventIDCode.2083');
		2084 :  AlarmCount[29 ] := AlarmCount[29]  + 1;   MpAlarmXSet(AlarmMpLink,'EventIDCode.2084');
		2085 :  AlarmCount[30 ] := AlarmCount[30]  + 1;   MpAlarmXSet(AlarmMpLink,'EventIDCode.2085');
		2090 :  AlarmCount[31 ] := AlarmCount[31]  + 1;   MpAlarmXSet(AlarmMpLink,'EventIDCode.2090');
		2091 :  AlarmCount[32 ] := AlarmCount[32]  + 1;   MpAlarmXSet(AlarmMpLink,'EventIDCode.2091');
		2092 :  AlarmCount[33 ] := AlarmCount[33]  + 1;   MpAlarmXSet(AlarmMpLink,'EventIDCode.2092');
		2093 :  AlarmCount[34 ] := AlarmCount[34]  + 1;   MpAlarmXSet(AlarmMpLink,'EventIDCode.2093');
		2094 :  AlarmCount[35 ] := AlarmCount[35]  + 1;   MpAlarmXSet(AlarmMpLink,'EventIDCode.2094');
		2095 :  AlarmCount[36 ] := AlarmCount[36]  + 1;   MpAlarmXSet(AlarmMpLink,'EventIDCode.2095');
		2097 :  AlarmCount[37 ] := AlarmCount[37]  + 1;   MpAlarmXSet(AlarmMpLink,'EventIDCode.2097');
		2098 :  AlarmCount[38 ] := AlarmCount[38]  + 1;   MpAlarmXSet(AlarmMpLink,'EventIDCode.2098');
		2099 :  AlarmCount[39 ] := AlarmCount[39]  + 1;   MpAlarmXSet(AlarmMpLink,'EventIDCode.2099');
		2100 :  AlarmCount[40 ] := AlarmCount[40]  + 1;   MpAlarmXSet(AlarmMpLink,'EventIDCode.2100');
		2101 :  AlarmCount[41 ] := AlarmCount[41]  + 1;   MpAlarmXSet(AlarmMpLink,'EventIDCode.2101');
		2102 :  AlarmCount[42 ] := AlarmCount[42]  + 1;   MpAlarmXSet(AlarmMpLink,'EventIDCode.2102');
		2103 :  AlarmCount[43 ] := AlarmCount[43]  + 1;   MpAlarmXSet(AlarmMpLink,'EventIDCode.2103');
		2104 :  AlarmCount[44 ] := AlarmCount[44]  + 1;   MpAlarmXSet(AlarmMpLink,'EventIDCode.2104');
		2105 :  AlarmCount[45 ] := AlarmCount[45]  + 1;   MpAlarmXSet(AlarmMpLink,'EventIDCode.2105');
		2106 :  AlarmCount[46 ] := AlarmCount[46]  + 1;   MpAlarmXSet(AlarmMpLink,'EventIDCode.2106');
		2107 :  AlarmCount[47 ] := AlarmCount[47]  + 1;   MpAlarmXSet(AlarmMpLink,'EventIDCode.2107');
		2108 :  AlarmCount[48 ] := AlarmCount[48]  + 1;   MpAlarmXSet(AlarmMpLink,'EventIDCode.2108');
		2109 :  AlarmCount[49 ] := AlarmCount[49]  + 1;   MpAlarmXSet(AlarmMpLink,'EventIDCode.2109');
		2110 :  AlarmCount[50 ] := AlarmCount[50]  + 1;   MpAlarmXSet(AlarmMpLink,'EventIDCode.2110');
		2111 :  AlarmCount[51 ] := AlarmCount[51]  + 1;   MpAlarmXSet(AlarmMpLink,'EventIDCode.2111');
		2112 :  AlarmCount[52 ] := AlarmCount[52]  + 1;   MpAlarmXSet(AlarmMpLink,'EventIDCode.2112');
		4096 :  AlarmCount[53 ] := AlarmCount[53]  + 1;   MpAlarmXSet(AlarmMpLink,'EventIDCode.4096');
		4097 :  AlarmCount[54 ] := AlarmCount[54]  + 1;   MpAlarmXSet(AlarmMpLink,'EventIDCode.4097');
		4101 :  AlarmCount[55 ] := AlarmCount[55]  + 1;   MpAlarmXSet(AlarmMpLink,'EventIDCode.4101');
		4102 :  AlarmCount[56 ] := AlarmCount[56]  + 1;   MpAlarmXSet(AlarmMpLink,'EventIDCode.4102');
		6144 :  AlarmCount[57 ] := AlarmCount[57]  + 1;   MpAlarmXSet(AlarmMpLink,'EventIDCode.6144');
		6165 :  AlarmCount[58 ] := AlarmCount[58]  + 1;   MpAlarmXSet(AlarmMpLink,'EventIDCode.6165');
		6148 :  AlarmCount[59 ] := AlarmCount[59]  + 1;   MpAlarmXSet(AlarmMpLink,'EventIDCode.6148');
		6149 :  AlarmCount[60 ] := AlarmCount[60]  + 1;   MpAlarmXSet(AlarmMpLink,'EventIDCode.6149');
		6156 :  AlarmCount[61 ] := AlarmCount[61]  + 1;   MpAlarmXSet(AlarmMpLink,'EventIDCode.6156');
		6157 :  AlarmCount[62 ] := AlarmCount[62]  + 1;   MpAlarmXSet(AlarmMpLink,'EventIDCode.6157');
		6158 :  AlarmCount[63 ] := AlarmCount[63]  + 1;   MpAlarmXSet(AlarmMpLink,'EventIDCode.6158');
		12288:  AlarmCount[64 ] := AlarmCount[64]  + 1;   MpAlarmXSet(AlarmMpLink,'EventIDCode.12288');
		12291:  AlarmCount[65 ] := AlarmCount[65]  + 1;   MpAlarmXSet(AlarmMpLink,'EventIDCode.12291');
		12293:  AlarmCount[66 ] := AlarmCount[66]  + 1;   MpAlarmXSet(AlarmMpLink,'EventIDCode.12293');
		12294:  AlarmCount[67 ] := AlarmCount[67]  + 1;   MpAlarmXSet(AlarmMpLink,'EventIDCode.12294');
		12295:  AlarmCount[68 ] := AlarmCount[68]  + 1;   MpAlarmXSet(AlarmMpLink,'EventIDCode.12295');
		12296:  AlarmCount[69 ] := AlarmCount[69]  + 1;   MpAlarmXSet(AlarmMpLink,'EventIDCode.12296');
		12297:  AlarmCount[70 ] := AlarmCount[70]  + 1;   MpAlarmXSet(AlarmMpLink,'EventIDCode.12297');
		12298:  AlarmCount[71 ] := AlarmCount[71]  + 1;   MpAlarmXSet(AlarmMpLink,'EventIDCode.12298');
		12299:  AlarmCount[72 ] := AlarmCount[72]  + 1;   MpAlarmXSet(AlarmMpLink,'EventIDCode.12299');
		12300:  AlarmCount[73 ] := AlarmCount[73]  + 1;   MpAlarmXSet(AlarmMpLink,'EventIDCode.12300');
		12301:  AlarmCount[74 ] := AlarmCount[74]  + 1;   MpAlarmXSet(AlarmMpLink,'EventIDCode.12301');
		12302:  AlarmCount[75 ] := AlarmCount[75]  + 1;   MpAlarmXSet(AlarmMpLink,'EventIDCode.12302');
		12303:  AlarmCount[76 ] := AlarmCount[76]  + 1;   MpAlarmXSet(AlarmMpLink,'EventIDCode.12303');
		12304:  AlarmCount[77 ] := AlarmCount[77]  + 1;   MpAlarmXSet(AlarmMpLink,'EventIDCode.12304');
		12305:  AlarmCount[78 ] := AlarmCount[78]  + 1;   MpAlarmXSet(AlarmMpLink,'EventIDCode.12305');
		12307:  AlarmCount[79 ] := AlarmCount[79]  + 1;   MpAlarmXSet(AlarmMpLink,'EventIDCode.12307');
		12312:  AlarmCount[80 ] := AlarmCount[80]  + 1;   MpAlarmXSet(AlarmMpLink,'EventIDCode.12312');
		12313:  AlarmCount[81 ] := AlarmCount[81]  + 1;   MpAlarmXSet(AlarmMpLink,'EventIDCode.12313');
		12314:  AlarmCount[82 ] := AlarmCount[82]  + 1;   MpAlarmXSet(AlarmMpLink,'EventIDCode.12314');
		12315:  AlarmCount[83 ] := AlarmCount[83]  + 1;   MpAlarmXSet(AlarmMpLink,'EventIDCode.12315');
		12316:  AlarmCount[84 ] := AlarmCount[84]  + 1;   MpAlarmXSet(AlarmMpLink,'EventIDCode.12316');
		12317:  AlarmCount[85 ] := AlarmCount[85]  + 1;   MpAlarmXSet(AlarmMpLink,'EventIDCode.12317');
		12320:  AlarmCount[86 ] := AlarmCount[86]  + 1;   MpAlarmXSet(AlarmMpLink,'EventIDCode.12320');
		12322:  AlarmCount[87 ] := AlarmCount[87]  + 1;   MpAlarmXSet(AlarmMpLink,'EventIDCode.12322');
		12323:  AlarmCount[88 ] := AlarmCount[88]  + 1;   MpAlarmXSet(AlarmMpLink,'EventIDCode.12323');
		12328:  AlarmCount[89 ] := AlarmCount[89]  + 1;   MpAlarmXSet(AlarmMpLink,'EventIDCode.12328');
		12330:  AlarmCount[90 ] := AlarmCount[90]  + 1;   MpAlarmXSet(AlarmMpLink,'EventIDCode.12330');
		12331:  AlarmCount[91 ] := AlarmCount[91]  + 1;   MpAlarmXSet(AlarmMpLink,'EventIDCode.12331');
		12333:  AlarmCount[92 ] := AlarmCount[92]  + 1;   MpAlarmXSet(AlarmMpLink,'EventIDCode.12333');
		12334:  AlarmCount[93 ] := AlarmCount[93]  + 1;   MpAlarmXSet(AlarmMpLink,'EventIDCode.12334');
		12335:  AlarmCount[94 ] := AlarmCount[94]  + 1;   MpAlarmXSet(AlarmMpLink,'EventIDCode.12335');
		12336:  AlarmCount[95 ] := AlarmCount[95]  + 1;   MpAlarmXSet(AlarmMpLink,'EventIDCode.12336');
		12337:  AlarmCount[96 ] := AlarmCount[96]  + 1;   MpAlarmXSet(AlarmMpLink,'EventIDCode.12337');
		12338:  AlarmCount[97 ] := AlarmCount[97]  + 1;   MpAlarmXSet(AlarmMpLink,'EventIDCode.12338');
		12340:  AlarmCount[98 ] := AlarmCount[98]  + 1;   MpAlarmXSet(AlarmMpLink,'EventIDCode.12340');
		12341:  AlarmCount[99 ] := AlarmCount[99]  + 1;   MpAlarmXSet(AlarmMpLink,'EventIDCode.12341');
		12342:  AlarmCount[100] := AlarmCount[100] + 1;   MpAlarmXSet(AlarmMpLink,'EventIDCode.12342');
		12343:  AlarmCount[101] := AlarmCount[101] + 1;   MpAlarmXSet(AlarmMpLink,'EventIDCode.12343');
		12344:  AlarmCount[102] := AlarmCount[102] + 1;   MpAlarmXSet(AlarmMpLink,'EventIDCode.12344');
		12345:  AlarmCount[103] := AlarmCount[103] + 1;   MpAlarmXSet(AlarmMpLink,'EventIDCode.12345');
		12346:  AlarmCount[104] := AlarmCount[104] + 1;   MpAlarmXSet(AlarmMpLink,'EventIDCode.12346');
		12347:  AlarmCount[105] := AlarmCount[105] + 1;   MpAlarmXSet(AlarmMpLink,'EventIDCode.12347');
		12348:  AlarmCount[106] := AlarmCount[106] + 1;   MpAlarmXSet(AlarmMpLink,'EventIDCode.12348');
		4007:   AlarmCount[107] := AlarmCount[107] + 1;   MpAlarmXSet(AlarmMpLink,'EventIDCode.4007');
		7230:   AlarmCount[108] := AlarmCount[108] + 1;   MpAlarmXSet(AlarmMpLink,'EventIDCode.7230');
		4005:   AlarmCount[109] := AlarmCount[109] + 1;   MpAlarmXSet(AlarmMpLink,'EventIDCode.4005');
		4098:   AlarmCount[110] := AlarmCount[110] + 1;   MpAlarmXSet(AlarmMpLink,'EventIDCode.4098');
		9106:   AlarmCount[111] := AlarmCount[111] + 1;   MpAlarmXSet(AlarmMpLink,'EventIDCode.9106');

		ELSE
			MpAlarmXSet(AlarmMpLink,'EventIDCode.xxxx');
		END_CASE

END_FUNCTION
```

#### Main.st
```iecst
// --------------------------------------------------------------------------------------------------------------------
// Logbook Task
// This task reads the PLC logbook and creates the data structure to display it in mappView
// --------------------------------------------------------------------------------------------------------------------
PROGRAM _INIT
	// Set time range to all on startup
	DTGetTime_0.enable := TRUE;
	DTGetTime_0();
	LogbookInterface.Par.FilterDateStart := STRING_TO_DATE('D#1999-12-31');
	LogbookInterface.Par.FilterDateEnd := DT_TO_DATE(DTGetTime_0.DT1);

	// Read data after reboot
	LogbookInterface.Cmd.Refresh := TRUE;

	// define what object type should be searched for
	LogbookInterface.SegError.ParaSegFilter		:= 'gSeg_';
END_PROGRAM

PROGRAM _CYCLIC
	// Abort current update run
	IF EDGENEG(LogbookInterface.Cmd.Refresh) THEN
		IF 	LogbookState <> STATE_ERROR THEN
			LogbookInterface.Status := ERR_OK;
			LogbookState := STATE_WAIT;
		END_IF
	END_IF

	IF EDGEPOS(DiagInterface.TrakInterface.Asm.Status.ErrorStop) THEN
		LogbookInterface.Cmd.Update := TRUE;
	END_IF

	// Run task multiple times to speed up process
	FOR executions:=1 TO LOGBOOK_EXECUTIONS DO
		// --------------------------------------------------------------------------------------------------------------------
		// Logbook State machine
		// --------------------------------------------------------------------------------------------------------------------
		CASE LogbookState OF
		// --------------------------------------------------------------------------------------------------------------------
		// Wait for new command
		// --------------------------------------------------------------------------------------------------------------------
			STATE_WAIT:
				// --------------------------------------------------------------------------------------------------------------------
				// Get current date
				DTGetTime_0.enable := TRUE;
				DTGetTime_0();
				LogbookInterface.Par.DateNow := DTGetTime_0.DT1;
				LogbookInterface.Par.EntriesMax := LOGBOOK_ENTRIES_MAX;

				// --------------------------------------------------------------------------------------------------------------------
				// Refresh all logbook data
				IF LogbookInterface.Cmd.Refresh THEN
					// Erase old data, set busy state
					brsmemset(ADR(Logbook), 0, SIZEOF(Logbook));
					brsmemset(ADR(LogbookInterface.Data), 0, SIZEOF(LogbookInterface.Data));
					LogbookInterface.Status := ERR_FUB_BUSY;
					LogbookState := STATE_OPEN;
				END_IF

				// --------------------------------------------------------------------------------------------------------------------
				// Auto update logbook data
				IF LogbookInterface.Par.AutoUpdate THEN
					AutoRefresh.IN := TRUE;
					AutoRefresh.PT := LogbookInterface.Par.AutoUpdateInterval*100;
					AutoRefresh();
					IF AutoRefresh.Q THEN
						AutoRefresh(IN:= FALSE);
						LogbookInterface.Cmd.Update := TRUE;
						LogbookState := STATE_NEXT;
					END_IF
				ELSE
					AutoRefresh(IN:= FALSE);
				END_IF

				// --------------------------------------------------------------------------------------------------------------------
				// Update only latest logbook data
				IF LogbookInterface.Cmd.Update THEN
					brsmemset(ADR(Logbook.RecordIDIsLast), 0, SIZEOF(Logbook.RecordIDIsLast));
					brsmemset(ADR(Logbook.RecordID), 0, SIZEOF(Logbook.RecordID));

					brsmemset(ADR(LogbookInterface.SegError.Record), 0, SIZEOF(LogbookInterface.SegError.Record));
					LogbookInterface.SegError.Message := '';
					SegmentErrorFound := 0;

					brsmemset(ADR(AlarmCount), 0, SIZEOF(AlarmCount));

					// Start at the beginning set busy state
					Logbook.CntLogbook := 0;
					LogbookInterface.Status := ERR_FUB_BUSY;
					LogbookState := STATE_LATEST;
				END_IF

				// --------------------------------------------------------------------------------------------------------------------
				// Create new logbook entry
				IF LogbookInterface.Cmd.Create THEN
					LogbookInterface.Status := ERR_FUB_BUSY;
					LogbookState := STATE_CREATE;
				END_IF

				// --------------------------------------------------------------------------------------------------------------------
				// Reset function blocks
				ArEventLogGetIdent_0(Execute := FALSE);
				ArEventLogGetLatestRecordID_0(Execute := FALSE);
				ArEventLogGetPreviousRecordID_0(Execute := FALSE);
				ArEventLogRead_0(Execute := FALSE);
				ArEventLogReadErrorNumber_0(Execute := FALSE);
				ArEventLogReadDescription_0(Execute := FALSE);
				ArEventLogReadAddData_0(Execute := FALSE);
				ArEventLogWrite_0(Execute := FALSE);
				ArEventLogReadObjectID_0(Execute := FALSE);

				// --------------------------------------------------------------------------------------------------------------------
				// Show status, reset error command
				LogbookInterface.Cmd.ResetError := FALSE;
				LogbookInterface.StatusText := 'Waiting...last update ';
				brsstrcat(ADR(LogbookInterface.StatusText), ADR(LogbookInterface.Data.LastUpdate));
				EXIT;
		// --------------------------------------------------------------------------------------------------------------------
		// Create a new logbook entry
		// --------------------------------------------------------------------------------------------------------------------
			STATE_CREATE:
				eventID := ArEventLogMakeEventID(UDINT_TO_USINT(LogbookInterface.Par.CreateSeverity), 0 , LogbookInterface.Par.CreateErrorNo);
				brsmemset(ADR(AddData), 0, SIZEOF(AddData));
				brsstrcpy(ADR(AddData), ADR(LogbookInterface.Par.CreateErrorText));

				ArEventLogWrite_0.Execute := TRUE;
				ArEventLogWrite_0.Ident := Logbook.Ident[LogbookInterface.Par.CreateLogbook];
				ArEventLogWrite_0.EventID := eventID;
				ArEventLogWrite_0.ObjectID := 'User event';
				ArEventLogWrite_0.AddDataFormat := arEVENTLOG_ADDFORMAT_TEXT;
				ArEventLogWrite_0.AddData := ADR(AddData);
				ArEventLogWrite_0.AddDataSize := brsstrlen(ADR(AddData));
				ArEventLogWrite_0();

				// Success
				IF ArEventLogWrite_0.Done AND ArEventLogWrite_0.StatusID = ERR_OK THEN
					ArEventLogWrite_0(Execute := FALSE);
					LogbookInterface.Cmd.Create := FALSE;
					LogbookInterface.Cmd.Update := TRUE;
					LogbookState := STATE_WAIT;
				// Error
				ELSIF ArEventLogWrite_0.Error THEN
					LogbookInterface.Error.State := LogbookState;
					LogbookInterface.Status := ArEventLogWrite_0.StatusID;
					LogbookState := STATE_ERROR;
				END_IF
		// --------------------------------------------------------------------------------------------------------------------
		// Open logbook
		// --------------------------------------------------------------------------------------------------------------------
			STATE_OPEN:
				// Last logbook reached
				IF Logbook.CntLogbook > LOGBOOK_BOOKS_MAX THEN
					Logbook.CntLogbook := 0;
					LogbookState := STATE_LATEST;
					EXIT;
				END_IF
				ArEventLogGetIdent_0.Execute := LogbookInterface.Cmd.Refresh;
				ArEventLogGetIdent_0.Name := LOGBOOK_NAMES[Logbook.CntLogbook];
				ArEventLogGetIdent_0();

				// Success
				IF (ArEventLogGetIdent_0.Done AND ArEventLogGetIdent_0.StatusID = ERR_OK) OR ArEventLogGetIdent_0.StatusID = arEVENTLOG_ERR_LOGBOOK_NOT_FOUND THEN
					Logbook.Ident[Logbook.CntLogbook] := ArEventLogGetIdent_0.Ident;
					Logbook.CntLogbook := Logbook.CntLogbook + 1;
					ArEventLogGetIdent_0(Execute := FALSE);
					// Error
				ELSIF ArEventLogGetIdent_0.Error THEN
					LogbookInterface.Error.State := LogbookState;
					LogbookInterface.Status := ArEventLogGetIdent_0.StatusID;
					LogbookState := STATE_ERROR;
				END_IF
		// --------------------------------------------------------------------------------------------------------------------
		// Read latest entry
		// --------------------------------------------------------------------------------------------------------------------
			STATE_LATEST:
				ArEventLogGetLatestRecordID_0.Execute := TRUE;
				ArEventLogGetLatestRecordID_0.Ident := Logbook.Ident[Logbook.CntLogbook];
				ArEventLogGetLatestRecordID_0();

				// Success
				IF ArEventLogGetLatestRecordID_0.Done AND ArEventLogGetLatestRecordID_0.StatusID = ERR_OK THEN
					// Store this record ID for next step
					Logbook.RecordID[Logbook.CntLogbook] := ArEventLogGetLatestRecordID_0.RecordID;
					// If there is a new entry
					IF ArEventLogGetLatestRecordID_0.RecordID > Logbook.RecordIDOld[Logbook.CntLogbook] THEN
						// Store latest ID for next update command, reset is last flag
						Logbook.RecordIDLatest[Logbook.CntLogbook] := ArEventLogGetLatestRecordID_0.RecordID;
						LogbookState := STATE_DETAILS_1;
						// No new entry
					ELSE
						Logbook.RecordIDIsLast[Logbook.CntLogbook] := TRUE;
						LogbookState := STATE_PREP;
					END_IF
					// Error
				ELSIF ArEventLogGetLatestRecordID_0.Error THEN
					LogbookInterface.Error.State := LogbookState;
					LogbookInterface.Status := ArEventLogGetLatestRecordID_0.StatusID;
					LogbookState := STATE_ERROR;
				END_IF
		// --------------------------------------------------------------------------------------------------------------------
		// Read next entry
		// --------------------------------------------------------------------------------------------------------------------
			STATE_NEXT:
				animation := WorkingStatus(ADR(LogbookInterface.StatusText), ADR('reading entries...'), animation);
				ArEventLogGetPreviousRecordID_0.Execute := TRUE;
				ArEventLogGetPreviousRecordID_0.Ident := Logbook.Ident[Logbook.CntLogbook];
				ArEventLogGetPreviousRecordID_0.RecordID := Logbook.RecordID[Logbook.CntLogbook];
				ArEventLogGetPreviousRecordID_0();

				// Success
				IF ArEventLogGetPreviousRecordID_0.Done AND ArEventLogGetPreviousRecordID_0.StatusID = ERR_OK THEN
					// Store this record ID for next step
					Logbook.RecordID[Logbook.CntLogbook] := ArEventLogGetPreviousRecordID_0.PrevRecordID;
					// Stop update when previous record ID is reached
					IF Logbook.RecordID[Logbook.CntLogbook] = Logbook.RecordIDOld[Logbook.CntLogbook] AND LogbookInterface.Cmd.Update THEN
						// Remember latest entry, set is last flag
						Logbook.RecordIDOld[Logbook.CntLogbook] := Logbook.RecordIDLatest[Logbook.CntLogbook];
						Logbook.RecordIDIsLast[Logbook.CntLogbook] := TRUE;
						LogbookState := STATE_PREP;
					ELSE
						LogbookState := STATE_DETAILS_1;
					END_IF
					// Error
				ELSIF ArEventLogGetPreviousRecordID_0.Error THEN
					// Last entry reached is not an error
					IF ArEventLogGetPreviousRecordID_0.StatusID = arEVENTLOG_ERR_RECORDID_INVALID THEN
						// Remember latest entry, set is last flag
						Logbook.RecordIDOld[Logbook.CntLogbook] := Logbook.RecordIDLatest[Logbook.CntLogbook];
						Logbook.RecordIDIsLast[Logbook.CntLogbook] := TRUE;
						LogbookState := STATE_PREP;
						// Everything else is an error
					ELSE
						LogbookInterface.Error.State := LogbookState;
						LogbookInterface.Status := ArEventLogGetPreviousRecordID_0.StatusID;
						LogbookState := STATE_ERROR;
					END_IF
				END_IF
		// --------------------------------------------------------------------------------------------------------------------
		// Read event id and time stamp
		// --------------------------------------------------------------------------------------------------------------------
			STATE_DETAILS_1:
				ArEventLogRead_0.Execute := TRUE;
				ArEventLogRead_0.Ident := Logbook.Ident[Logbook.CntLogbook];
				ArEventLogRead_0.RecordID := Logbook.RecordID[Logbook.CntLogbook];
				ArEventLogRead_0();

				// Success
				IF ArEventLogRead_0.Done AND (ArEventLogRead_0.StatusID = ERR_OK OR ArEventLogRead_0.StatusID = arEVENTLOG_WRN_NO_EVENTID) THEN
					LogbookState := STATE_DETAILS_2;

					EventID := ArEventLogRead_0.EventID;
					EventTimeStamp := ArEventLogRead_0.TimeStamp;
					EventIDSeverity	:= DINT_TO_USINT(SHR(EventID, 30) AND 16#03);
					EventIDFacility	:= DINT_TO_UINT(SHR(EventID, 16) AND 16#0FFF);
					EventIDCode		:= DINT_TO_UINT(SHR(EventID, 0) AND 16#FFFF);

				// Error
				ELSIF ArEventLogRead_0.Error THEN
					LogbookInterface.Error.State := LogbookState;
					LogbookInterface.Status := ArEventLogRead_0.StatusID;
					LogbookState := STATE_ERROR;
				END_IF
		// --------------------------------------------------------------------------------------------------------------------
		// Read error no
		// --------------------------------------------------------------------------------------------------------------------
			STATE_DETAILS_2:
				ArEventLogReadErrorNumber_0.Execute := TRUE;
				ArEventLogReadErrorNumber_0.Ident := Logbook.Ident[Logbook.CntLogbook];
				ArEventLogReadErrorNumber_0.RecordID := Logbook.RecordID[Logbook.CntLogbook];
				ArEventLogReadErrorNumber_0();

				// Success
				IF (ArEventLogReadErrorNumber_0.Done AND ArEventLogReadErrorNumber_0.StatusID = ERR_OK) OR ArEventLogReadErrorNumber_0.StatusID = arEVENTLOG_ERR_NO_ERRORNUMBER THEN
					brsmemset(ADR(ErrorText), 0, SIZEOF(ErrorText));
					LogbookState := STATE_DETAILS_3;
				// Error
				ELSIF ArEventLogReadErrorNumber_0.Error THEN
					LogbookInterface.Error.State := LogbookState;
					LogbookInterface.Status := ArEventLogReadErrorNumber_0.StatusID;
					LogbookState := STATE_ERROR;
				END_IF
		// --------------------------------------------------------------------------------------------------------------------
		// Read error description
		// --------------------------------------------------------------------------------------------------------------------
			STATE_DETAILS_3:
				ArEventLogReadDescription_0.Execute := TRUE;
				ArEventLogReadDescription_0.Ident := Logbook.Ident[Logbook.CntLogbook];
				ArEventLogReadDescription_0.RecordID := Logbook.RecordID[Logbook.CntLogbook];
				ArEventLogReadDescription_0.TextBuffer := ADR(ErrorText);
				ArEventLogReadDescription_0.TextBufferSize := SIZEOF(ErrorText);
				ArEventLogReadDescription_0();

				// Success
				IF (ArEventLogReadDescription_0.Done AND (ArEventLogReadDescription_0.StatusID = ERR_OK OR ArEventLogReadDescription_0.StatusID = arEVENTLOG_WRN_NO_EVENTID)) OR ArEventLogReadDescription_0.StatusID = arEVENTLOG_ERR_NO_DESCRIPTION THEN
					brsmemset(ADR(AddData), 0, SIZEOF(AddData));
					IF ((Logbook.CntLogbook = 6) AND (EventIDSeverity = arEVENTLOG_SEVERITY_ERROR)) THEN (*6 = index for motion logbook*)
						LogbookState := STATE_CHECK_FILTER;
					ELSE
						LogbookState := STATE_DETAILS_4;
					END_IF
				// Error
				ELSIF ArEventLogReadDescription_0.Error THEN
					LogbookInterface.Error.State := LogbookState;
					LogbookInterface.Status := ArEventLogReadDescription_0.StatusID;
					LogbookState := STATE_ERROR;
				END_IF
		// --------------------------------------------------------------------------------------------------------------------
		// Check if 'Error' has been entered by a Segment
		// --------------------------------------------------------------------------------------------------------------------
			STATE_CHECK_FILTER:
				ArEventLogReadObjectID_0.Execute	:= TRUE;
				ArEventLogReadObjectID_0.Ident		:= Logbook.Ident[Logbook.CntLogbook];
				ArEventLogReadObjectID_0.RecordID	:= Logbook.RecordID[Logbook.CntLogbook];
				ArEventLogReadObjectID_0();

				IF ArEventLogReadObjectID_0.Done THEN
					ObjectID := ArEventLogReadObjectID_0.ObjectID;
					ArEventLogReadObjectID_0.Execute := FALSE;
					IF brsmemcmp(ADR(ObjectID), ADR(LogbookInterface.SegError.ParaSegFilter), 3) = 0 THEN
						LogbookState := STATE_UPDATE_LIST;
					ELSE
						LogbookState := STATE_DETAILS_4;
					END_IF
				ELSIF ArEventLogReadObjectID_0.Error THEN
					LogbookInterface.SegError.Message := 'Error ReadObjectID';
					LogbookState := STATE_ERROR;
				END_IF

		// --------------------------------------------------------------------------------------------------------------------
		// Update the segment error list which is used for alarms
		// --------------------------------------------------------------------------------------------------------------------
			STATE_UPDATE_LIST:
				LogbookInterface.SegError.Record[SegmentErrorFound].ObjectID		:= ObjectID;
				LogbookInterface.SegError.Record[SegmentErrorFound].EventID			:= EventID;
				LogbookInterface.SegError.Record[SegmentErrorFound].EventIDSeverity	:= EventIDSeverity;
				LogbookInterface.SegError.Record[SegmentErrorFound].EventIDFacility	:= EventIDFacility;
				LogbookInterface.SegError.Record[SegmentErrorFound].EventIDCode		:= EventIDCode;
				LogbookInterface.SegError.Record[SegmentErrorFound].Description		:= Description;

				LogbookInterface.SegError.Record[SegmentErrorFound].EventTimeStamp	:= UDINT_TO_TIME((EventTimeStamp.sec MOD (24*60*60))*1000 + (EventTimeStamp.nsec / 1000000));		// convert to TIME format (ms since start of day)

				brsstrcpy(ADR(LogbookInterface.SegError.Record[SegmentErrorFound].Text), ADR(''));
				ascTIME(LogbookInterface.SegError.Record[SegmentErrorFound].EventTimeStamp, ADR(TempString), SIZEOF(TempString));
				TIME_TO_TIMEStructure(LogbookInterface.SegError.Record[SegmentErrorFound].EventTimeStamp,ADR(TimeStruct)); // for checking against older entries

				brsstrcat(ADR(LogbookInterface.SegError.Record[SegmentErrorFound].Text), ADR(TempString));
				brsstrcat(ADR(LogbookInterface.SegError.Record[SegmentErrorFound].Text), ADR(' => '));

				brsstrcat(ADR(LogbookInterface.SegError.Record[SegmentErrorFound].Text), ADR(ObjectID));

				brsstrcat(ADR(LogbookInterface.SegError.Record[SegmentErrorFound].Text), ADR(': Error '));
				brsitoa(EventIDCode, ADR(TempString));
				brsstrcat(ADR(LogbookInterface.SegError.Record[SegmentErrorFound].Text), ADR(TempString));

				brsstrcat(ADR(LogbookInterface.SegError.Record[SegmentErrorFound].Text), ADR(' => '));
				brsstrcat(ADR(LogbookInterface.SegError.Record[SegmentErrorFound].Text), ADR(Description));

				IF SegmentErrorFound = 0 THEN
					FirstEntryCheckSum := TimeStruct.minute; // save the timestamp minute of the first entry as checksum
				END_IF

				SegmentErrorFound := SegmentErrorFound + 1;

				SetTrakSegAlarm(DiagInterface.AlarmCore,EventIDCode,ADR(AlarmCount));

				// stop reading the logger when the end of the array is reached OR
				// when the entries start having a different timestamp which means they are older
				IF SegmentErrorFound > 499 OR (FirstEntryCheckSum <> (TimeStruct.minute) ) THEN
					LogbookState := STATE_DETAILS_4;
				ELSE
					LogbookState := STATE_DETAILS_4;
				END_IF

		// --------------------------------------------------------------------------------------------------------------------
		// Read additional information
		// --------------------------------------------------------------------------------------------------------------------
			STATE_DETAILS_4:
				// Skip if no additional data is available
				IF ArEventLogRead_0.AddDataSize > 0 THEN
					// Read additional data
					ArEventLogReadAddData_0.Execute := TRUE;
					ArEventLogReadAddData_0.Ident := Logbook.Ident[Logbook.CntLogbook];
					ArEventLogReadAddData_0.RecordID := Logbook.RecordID[Logbook.CntLogbook];
					ArEventLogReadAddData_0.AddData := ADR(AddData);
					// Limit buffer to max size
					IF ArEventLogRead_0.AddDataSize < SIZEOF(AddData) THEN
						ArEventLogReadAddData_0.BytesToRead := ArEventLogRead_0.AddDataSize;
					ELSE
						ArEventLogReadAddData_0.BytesToRead := SIZEOF(AddData);
					END_IF
					ArEventLogReadAddData_0();

					// Success
					IF (ArEventLogReadAddData_0.Done AND ArEventLogReadAddData_0.StatusID = ERR_OK) OR ArEventLogReadAddData_0.StatusID = arEVENTLOG_INF_SIZE THEN
						// Enter standard text if additional does not fit
						IF ArEventLogReadAddData_0.StatusID = arEVENTLOG_INF_SIZE THEN
							brsstrcat(ADR(ErrorText), ADR('\n >>> '));
							brsstrcat(ADR(ErrorText), ADR('Additional buffer is too small'));
						ELSE
							// Make sure string is readable
							IF brsstrcmp(ADR(AddData), ADR('')) <> 0 AND ArEventLogRead_0.AddDataFormat = arEVENTLOG_ADDFORMAT_TEXT THEN
								brsstrcat(ADR(ErrorText), ADR('\n >>> '));
								// Limit additional text to max size
								IF ArEventLogReadAddData_0.AddDataSize < SIZEOF(ErrorText) - brsstrlen(ADR(ErrorText)) THEN
									brsstrcat(ADR(ErrorText), ADR(AddData));
								ELSE
									brsmemcpy(ADR(ErrorText) + brsstrlen(ADR(ErrorText)), ADR(AddData), SIZEOF(ErrorText) - brsstrlen(ADR(ErrorText)));
								END_IF
							END_IF
						END_IF
						LogbookState := STATE_FILTER;
					// Error
					ELSIF ArEventLogReadDescription_0.Error THEN
						LogbookInterface.Error.State := LogbookState;
						LogbookInterface.Status := ArEventLogReadAddData_0.StatusID;
						LogbookState := STATE_ERROR;
					END_IF
				ELSE
					LogbookState := STATE_FILTER;
				END_IF
		// --------------------------------------------------------------------------------------------------------------------
		// Apply filter settings
		// --------------------------------------------------------------------------------------------------------------------
			STATE_FILTER:
				// --------------------------------------------------------------------------------------------------------------------
				// Filters
				cntFilterNo := 0;
				cntFilterText := 0;
				cntFilterLogbook := 0;
				cntFilterSeverity := 0;
				cntFilterDate := 0;
				// --------------------------------------------------------------------------------------------------------------------
				// Check if logbook should be read
				IF  LogbookInterface.Par.FilterLogbook[Logbook.CntLogbook] THEN
					cntFilterLogbook := cntFilterLogbook + 1;
				END_IF
				// --------------------------------------------------------------------------------------------------------------------
				// Check if error text matches search string
				IF LogbookInterface.Par.FilterErrorText = '' OR IsInstr(ADR(ErrorText), ADR(LogbookInterface.Par.FilterErrorText)) THEN
					cntFilterText := cntFilterText + 1;
				END_IF
				// --------------------------------------------------------------------------------------------------------------------
				// Make sure error number matches filter
				IF LogbookInterface.Par.FilterErrorNo = 0 OR LogbookInterface.Par.FilterErrorNo = ArEventLogReadErrorNumber_0.ErrorNumber THEN
					cntFilterNo := cntFilterNo + 1;
				END_IF
				// --------------------------------------------------------------------------------------------------------------------
				// Check severity filter settings
				IF ArEventLogRead_0.EventID <> 0 THEN
					LogbookInterface.Data.CntSeverity[GetSeverity(EventID := ArEventLogRead_0.EventID)] := LogbookInterface.Data.CntSeverity[GetSeverity(EventID := ArEventLogRead_0.EventID)] + 1;
					IF LogbookInterface.Par.FilterSeverity[GetSeverity(EventID := ArEventLogRead_0.EventID)] THEN
						cntFilterSeverity := cntFilterSeverity + 1;
					END_IF
				ELSE
					LogbookInterface.Data.CntSeverity[ArEventLogReadErrorNumber_0.Severity] := LogbookInterface.Data.CntSeverity[ArEventLogReadErrorNumber_0.Severity] + 1;
					IF LogbookInterface.Par.FilterSeverity[ArEventLogReadErrorNumber_0.Severity] THEN
						cntFilterSeverity := cntFilterSeverity + 1;
					END_IF
				END_IF
				// --------------------------------------------------------------------------------------------------------------------
				// Check date range
				tmpSTR:= DT_TO_STRING(DATE_TO_DT(LogbookInterface.Par.FilterDateStart));
				brsmemcpy(ADR(tmpSTR)+13, ADR('-00:00:00'), 9);
				TimeStart := STRING_TO_DT(tmpSTR);
				tmpSTR:= DT_TO_STRING(DATE_TO_DT(LogbookInterface.Par.FilterDateEnd));
				brsmemcpy(ADR(tmpSTR)+13, ADR('-23:59:59'), 9);
				TimeEnd := STRING_TO_DT(tmpSTR);
				IF ArEventLogRead_0.TimeStamp.sec >= DT_TO_UDINT(TimeStart) AND ArEventLogRead_0.TimeStamp.sec <= DT_TO_UDINT(TimeEnd) THEN
					cntFilterDate := cntFilterDate + 1;
				END_IF
				// --------------------------------------------------------------------------------------------------------------------
				// Count logbook entries
				LogbookInterface.Data.CntLogbook[Logbook.CntLogbook] := LogbookInterface.Data.CntLogbook[Logbook.CntLogbook] +  1;

				// --------------------------------------------------------------------------------------------------------------------
				// Transfer data
				IF cntFilterNo > 0 AND cntFilterText > 0 AND cntFilterLogbook > 0 AND cntFilterSeverity > 0 AND cntFilterDate > 0 THEN
					// --------------------------------------------------------------------------------------------------------------------
					// Find new place for entry
					idx := InsertEntry(ADR(LogbookInterface.Data), ArEventLogRead_0.TimeStamp.sec, UDINT_TO_UINT(ArEventLogRead_0.TimeStamp.nsec/1000000), LogbookInterface.Par.Sorting);
					IF idx <> NO_SPACE THEN
						// Store date and time
						LogbookInterface.Data.Entries.DTsec[idx] := ArEventLogRead_0.TimeStamp.sec;
						LogbookInterface.Data.Entries.DTmsec[idx] := UDINT_TO_UINT(ArEventLogRead_0.TimeStamp.nsec/1000000);
						// Add timestamp
						tmpDT := UDINT_TO_DT(ArEventLogRead_0.TimeStamp.sec);
						DT_TO_DTStructure(tmpDT, ADR(tmpDTstruct));
						brsmemset(ADR(LogbookInterface.Data.Entries.Timestamp[idx]), 0, SIZEOF(LogbookInterface.Data.Entries.Timestamp[idx]));
						NormalizeDateTime(ADR(LogbookInterface.Data.Entries.Timestamp[idx]), tmpDTstruct.day, '');
						NormalizeDateTime(ADR(LogbookInterface.Data.Entries.Timestamp[idx]), tmpDTstruct.month, '.');
						NormalizeDateTime(ADR(LogbookInterface.Data.Entries.Timestamp[idx]), tmpDTstruct.year, '.');
						NormalizeDateTime(ADR(LogbookInterface.Data.Entries.Timestamp[idx]), tmpDTstruct.hour, ' ');
						NormalizeDateTime(ADR(LogbookInterface.Data.Entries.Timestamp[idx]), tmpDTstruct.minute, ':');
						NormalizeDateTime(ADR(LogbookInterface.Data.Entries.Timestamp[idx]), tmpDTstruct.second, ':');
						NormalizeDateTime(ADR(LogbookInterface.Data.Entries.Timestamp[idx]), LogbookInterface.Data.Entries.DTmsec[idx], '.');
						// Add event ID, code, logbook, severity
						LogbookInterface.Data.Entries.EventID[LogbookInterface.Data.EntriesTotal] := ArEventLogRead_0.EventID;
						IF ArEventLogRead_0.EventID <> 0 THEN
							LogbookInterface.Data.Entries.Severity[idx] := GetSeverity(EventID := ArEventLogRead_0.EventID);
						ELSE
							LogbookInterface.Data.Entries.Severity[idx] := ArEventLogReadErrorNumber_0.Severity;
						END_IF
						LogbookInterface.Data.Entries.Code[idx] := GetCode(EventID := ArEventLogRead_0.EventID);
						LogbookInterface.Data.Entries.FacilityCode[idx] := GetFacility(EventID := ArEventLogRead_0.EventID);
						LogbookInterface.Data.Entries.LogbookName[idx] := LOGBOOK_TEXT[Logbook.CntLogbook];
						// Add error number and text, use event ID if error no is 0
						IF ArEventLogReadErrorNumber_0.ErrorNumber <> 0 THEN
							LogbookInterface.Data.Entries.ErrorNo[idx] := ArEventLogReadErrorNumber_0.ErrorNumber;
						ELSE
							LogbookInterface.Data.Entries.ErrorNo[idx] := ArEventLogRead_0.EventID;
						END_IF
						httpUtf8ToString_0(enable := TRUE, pSrc := ADR(ErrorText), pDest := ADR(LogbookInterface.Data.Entries.ErrorText[idx]), destSize := SIZEOF(LogbookInterface.Data.Entries.ErrorText[idx]));
					END_IF
				END_IF

				// --------------------------------------------------------------------------------------------------------------------
				// Hide unused table rows
				brsitoa(LogbookInterface.Data.EntriesTotal, ADR(tmpSTR));
				LogbookInterface.Par.TableConfig := '{"specRows":[{"from":';
				brsstrcat(ADR(LogbookInterface.Par.TableConfig), ADR(tmpSTR));
				brsstrcat(ADR(LogbookInterface.Par.TableConfig), ADR(', "to":'));
				brsitoa(LOGBOOK_ENTRIES_MAX, ADR(tmpSTR));
				brsstrcat(ADR(LogbookInterface.Par.TableConfig), ADR(tmpSTR));
				brsstrcat(ADR(LogbookInterface.Par.TableConfig), ADR(', "visible":false}]}'));

				LogbookState := STATE_PREP;

		// --------------------------------------------------------------------------------------------------------------------
		// Perpare for next entry
		// --------------------------------------------------------------------------------------------------------------------
			STATE_PREP:
				// --------------------------------------------------------------------------------------------------------------------
				// Reset buffer and function blocks
				brsmemset(ADR(AddData), 0, SIZEOF(AddData));
				ArEventLogGetLatestRecordID_0(Execute := FALSE);
				ArEventLogGetPreviousRecordID_0(Execute := FALSE);
				ArEventLogRead_0(Execute := FALSE);
				ArEventLogReadErrorNumber_0(Execute := FALSE);
				ArEventLogReadDescription_0(Execute := FALSE);
				ArEventLogReadAddData_0(Execute := FALSE);
				ArEventLogReadObjectID_0(Execute := FALSE);

				// --------------------------------------------------------------------------------------------------------------------
				// Find next logbook from here to the end
				REPEAT
					Logbook.CntLogbook := Logbook.CntLogbook + 1;
					IF Logbook.CntLogbook <= LOGBOOK_BOOKS_MAX THEN
						IF (Logbook.Ident[Logbook.CntLogbook] <> 0 AND NOT Logbook.RecordIDIsLast[Logbook.CntLogbook]) OR (Logbook.Ident[Logbook.CntLogbook] <> 0 AND Logbook.RecordID[Logbook.CntLogbook] = 0) THEN
							EXIT;
						END_IF
					END_IF
					UNTIL Logbook.CntLogbook > LOGBOOK_BOOKS_MAX
				END_REPEAT;

				// --------------------------------------------------------------------------------------------------------------------
				// No logbook found, start at the beginning
				IF Logbook.CntLogbook > LOGBOOK_BOOKS_MAX THEN
					Logbook.CntLogbook := 0;
					// Find next logbook from start to the end
					REPEAT
						IF (Logbook.Ident[Logbook.CntLogbook] <> 0 AND NOT Logbook.RecordIDIsLast[Logbook.CntLogbook]) OR (Logbook.Ident[Logbook.CntLogbook] <> 0 AND Logbook.RecordID[Logbook.CntLogbook] = 0) THEN
							EXIT;
						END_IF
						Logbook.CntLogbook := Logbook.CntLogbook + 1;
						UNTIL Logbook.CntLogbook > LOGBOOK_BOOKS_MAX
					END_REPEAT;
				END_IF

				// --------------------------------------------------------------------------------------------------------------------
				// Finish when no logbook found or max entries is reached
				IF Logbook.CntLogbook > LOGBOOK_BOOKS_MAX OR (LogbookInterface.Par.AbortOnEntriesLimit AND LogbookInterface.Data.EntriesTotal = LOGBOOK_ENTRIES_MAX) THEN
					// Add last update
					DT_TO_DTStructure(LogbookInterface.Par.DateNow, ADR(tmpDTstruct));
					brsmemset(ADR(LogbookInterface.Data.LastUpdate), 0, SIZEOF(LogbookInterface.Data.LastUpdate));
					NormalizeDateTime(ADR(LogbookInterface.Data.LastUpdate), tmpDTstruct.day, '');
					NormalizeDateTime(ADR(LogbookInterface.Data.LastUpdate), tmpDTstruct.month, '.');
					NormalizeDateTime(ADR(LogbookInterface.Data.LastUpdate), tmpDTstruct.year, '.');
					NormalizeDateTime(ADR(LogbookInterface.Data.LastUpdate), tmpDTstruct.hour, ' ');
					NormalizeDateTime(ADR(LogbookInterface.Data.LastUpdate), tmpDTstruct.minute, ':');
					NormalizeDateTime(ADR(LogbookInterface.Data.LastUpdate), tmpDTstruct.second, ':');
					// Reset status and command
					LogbookInterface.Status := ERR_OK;
					LogbookInterface.Cmd.Refresh := FALSE;
					LogbookInterface.Cmd.Update := FALSE;
					LogbookState := STATE_WAIT;
				ELSE
					// Read latest entry
					IF Logbook.RecordID[Logbook.CntLogbook] = 0 THEN
						LogbookState := STATE_LATEST;
						// Read next entry
					ELSE
						LogbookState := STATE_NEXT;
					END_IF
				END_IF

		// --------------------------------------------------------------------------------------------------------------------
		// Error state
		// --------------------------------------------------------------------------------------------------------------------
			STATE_ERROR:
				LogbookInterface.StatusText := 'Error...';
				brsmemset(ADR(LogbookInterface.Cmd), 0, SIZEOF(LogbookInterface.Cmd)-1);
				// Reset error
				IF LogbookInterface.Cmd.ResetError THEN
					LogbookInterface.Error.State := STATE_NONE;
					LogbookInterface.Status := 0;
					LogbookInterface.Cmd.ResetError := FALSE;
					LogbookState := STATE_WAIT;
				END_IF
				EXIT;
		END_CASE;
	END_FOR;

END_PROGRAM
```

### TrackDiagGlobal.typ - not listed in the package file held
```iecst
(*Insert your comment here.*)

TYPE
	ErrorSegInfoType : 	STRUCT
		Error : USINT;
	END_STRUCT;
END_TYPE

(*LogBook def*)

TYPE
	LogBookStateEnum :
		( (*State machine*)
		STATE_WAIT,
		STATE_CREATE,
		STATE_OPEN,
		STATE_LATEST,
		STATE_NEXT,
		STATE_DETAILS_1,
		STATE_DETAILS_2,
		STATE_DETAILS_3,
		STATE_CHECK_FILTER,
		STATE_UPDATE_LIST,
		STATE_DETAILS_4,
		STATE_FILTER,
		STATE_PREP,
		STATE_ERROR,
		STATE_NONE
		);
	LogBookSeverityEnum :
		(
		SEVERITY_NOTIFICATION,
		SEVERITY_INFORMATION,
		SEVERITY_WARNING,
		SEVERITY_ERROR
		);
	LogBookTypeEnum :
		(
		LOG_ACCESS_SECURITY,
		LOG_COMMISIONING,
		LOG_CONNECTIVITY,
		LOG_FIELDBUS,
		LOG_FIREWALL,
		LOG_MAPP,
		LOG_MOTION,
		LOG_SAFETY,
		LOG_SYSTEM,
		LOG_TEXTSYSTEM,
		LOG_UNITSYSTEM,
		LOG_USER,
		LOG_VISUALIZATION
		);
	LogBookSortingEnum :
		(
		SORTING_ASC,
		SORTING_DESC
		);
	LogBookParType : 	STRUCT  (*Parameter structure*)
		DateNow : DATE_AND_TIME; (*Current date and time*)
		TableConfig : STRING[100]; (*Hide unused rows*)
		EntriesMax : UINT; (*Maximum number of entries, shadow of LOGBOOK_ENTRIES_MAX*)
		FilterErrorNo : UDINT; (*Filter by error number*)
		FilterErrorText : STRING[LOGBOOK_TEXT_LEN]; (*Filter by error text*)
		FilterSeverity : ARRAY[0..3]OF BOOL := [4(TRUE)]; (*Filter by severity*)
		FilterLogbook : ARRAY[0..LOGBOOK_BOOKS_MAX]OF BOOL := [14(TRUE)]; (*Filter by logbook*)
		FilterDateStart : DATE; (*Filter by date*)
		FilterDateEnd : DATE;
		Sorting : LogBookSortingEnum := SORTING_DESC; (*Sort date asc or desc*)
		AbortOnEntriesLimit : BOOL; (*Stop looking for additional entries when limit is reached*)
		AutoUpdate : BOOL; (*Automatically update data*)
		AutoUpdateInterval : UINT := 60; (*Interval for auto update in s*)
		CreateErrorNo : UINT; (*Error no for new entry*)
		CreateErrorText : STRING[LOGBOOK_TEXT_LEN]; (*Error text for new entry*)
		CreateSeverity : LogBookSeverityEnum := SEVERITY_NOTIFICATION; (*Error severiry for new entry*)
		CreateLogbook : LogBookTypeEnum := LOG_USER; (*Error logbook for new entry*)
	END_STRUCT;
	LogBookErrorType : 	STRUCT  (*Error structure*)
		State : LogBookStateEnum; (*State where the error occured*)
	END_STRUCT;
	LogBookDataType : 	STRUCT  (*Data structure*)
		Entries : LogBookDataEntryType;
		EntriesTotal : UINT; (*Total number of entries*)
		CntSeverity : ARRAY[0..3]OF UINT; (*Counts by severity*)
		CntLogbook : ARRAY[0..LOGBOOK_BOOKS_MAX]OF UINT; (*Counts by logbook*)
		LastUpdate : STRING[25]; (*Last refresh run*)
	END_STRUCT;
	LogBookDataEntryType : 	STRUCT  (*Entries structure*)
		EventID : ARRAY[1..LOGBOOK_ENTRIES_MAX]OF DINT; (*Event ID*)
		Timestamp : ARRAY[1..LOGBOOK_ENTRIES_MAX]OF STRING[25]; (*Date and time*)
		DTsec : ARRAY[1..LOGBOOK_ENTRIES_MAX]OF UDINT; (*Date and time in sec*)
		DTmsec : ARRAY[1..LOGBOOK_ENTRIES_MAX]OF UDINT; (*Additional milliseconds*)
		Severity : ARRAY[1..LOGBOOK_ENTRIES_MAX]OF USINT; (*Severity*)
		Code : ARRAY[1..LOGBOOK_ENTRIES_MAX]OF UINT; (*Code*)
		FacilityCode : ARRAY[1..LOGBOOK_ENTRIES_MAX]OF UINT; (*Facility code*)
		LogbookName : ARRAY[1..LOGBOOK_ENTRIES_MAX]OF STRING[30]; (*Logbook text*)
		ErrorNo : ARRAY[1..LOGBOOK_ENTRIES_MAX]OF DINT; (*Error number*)
		ErrorText : ARRAY[1..LOGBOOK_ENTRIES_MAX]OF STRING[LOGBOOK_TEXT_LEN]; (*Error text*)
	END_STRUCT;
	LogBookCmdType : 	STRUCT  (*Command structure*)
		Refresh : BOOL; (*Read all entries*)
		Update : BOOL; (*Update entries*)
		Create : BOOL; (*Create a new entry*)
		ResetError : BOOL; (*Reset error*)
	END_STRUCT;
	LogBookSegErrorType : 	STRUCT
		ParaSegFilter : STRING[8]; (*show only entries with names beginning with this string*)
		Message : STRING[256]; (*message ArEventLog handling*)
		Record : ARRAY[0..500]OF LogBookSegErrorRecordType;
	END_STRUCT;
	LogBookSegErrorRecordType : 	STRUCT
		ObjectID : STRING[36]; (*logger entry "Entered by"*)
		EventID : DINT; (*logger entry "ID"*)
		EventIDSeverity : USINT; (*logger entry "Severity"*)
		EventIDFacility : UINT; (*logger entry "Facility"*)
		EventIDCode : UINT; (*logger entry "Code"*)
		EventTimeStamp : TIME; (*logger entry "Time"*)
		Text : STRING[300]; (*logger entry "Description"*)
		Description : STRING[256]; (*logger entry "Description"*)
	END_STRUCT;
	LogBookCtrlType : 	STRUCT  (*Main structure*)
		Cmd : LogBookCmdType;
		Par : LogBookParType;
		Data : LogBookDataType;
		Error : LogBookErrorType;
		SegError : LogBookSegErrorType;
		Status : DINT;
		StatusText : STRING[80];
	END_STRUCT;
END_TYPE
```

### TrackDiagGlobal.var - not listed in the package file held
```iecst
VAR CONSTANT
	NUM_HUBS : USINT := 5;
	NUM_PS : USINT := 5;
END_VAR
(*LogBook variables*)
VAR
	LogbookInterface : LogBookCtrlType; (*Logbook main structure*)
END_VAR
VAR CONSTANT
	LOGBOOK_EXECUTIONS : USINT := 10; (*Executions per cycle*)
	LOGBOOK_ENTRIES_MAX : UINT := 100; (*Total number of entries*)
	LOGBOOK_BOOKS_MAX : USINT := 13; (*Total number of facilities*)
	LOGBOOK_TEXT_LEN : UINT := 200; (*Error text length*)
END_VAR
(*Module definitions*)
VAR
	DiagInterface : ModuleInterfaceType;
	ModuleName : STRING[40];
END_VAR
```

### Program Logical/Source/Diagnostic/TrackDiag (IEC)

#### Init.st - Init, cyclic, exit code
```iecst
PROGRAM _INIT

	SegDefinition;

	paperCore.SegmentCount := TrackDiag.Seg.SegCount;
	paperCore.Segments := ADR(TrackDiag.Seg.SegList);
	paperCore.Options := ADR(paperOptions);
	paperCore.Enable := TRUE;
	paperCore.Assembly := ADR(DiagInterface.SampleTrak);
	paperCore.ShuttleMon := ADR(DiagInterface.ShuttleMon);

	//Replace with generated SVG ViewBox Values in format viewBox="MinX MinY Width Height"
	paperCore.ViewBoxCfg.MinX := -0.735577;
	paperCore.ViewBoxCfg.MinY := -0.115;
	paperCore.ViewBoxCfg.Width := 2.13115;
	paperCore.ViewBoxCfg.Height := 0.86;

END_PROGRAM
```
